C03649=1176.363,-28.044,-44.088,179.704,5.815,149.123
C03650=1176.358,-27.795,-44.101,179.705,5.815,149.122
C03651=1176.352,-27.545,-44.113,179.708,5.816,149.121
C03652=1176.347,-27.295,-44.125,179.711,5.816,149.121
C03653=1176.342,-27.046,-44.138,179.713,5.817,149.120
C03654=1176.337,-26.795,-44.150,179.715,5.817,149.120
C03655=1176.332,-26.546,-44.163,179.718,5.818,149.119
C03656=1176.327,-26.297,-44.175,179.720,5.819,149.118
C03657=1176.322,-26.047,-44.188,179.723,5.819,149.118
C03658=1176.316,-25.798,-44.200,179.725,5.819,149.117
C03659=1176.311,-25.548,-44.212,179.727,5.820,149.117
C03660=1176.307,-25.298,-44.225,179.730,5.820,149.116
C03661=1176.301,-25.048,-44.237,179.733,5.821,149.115
C03662=1176.296,-24.799,-44.250,179.735,5.821,149.115
C03663=1176.291,-24.550,-44.262,179.737,5.822,149.114
C03664=1176.286,-24.300,-44.275,179.740,5.822,149.113
C03665=1176.280,-24.030,-44.289,179.742,5.823,149.113
C03666=1176.275,-23.760,-44.302,179.745,5.824,149.112
C03667=1176.269,-23.491,-44.316,179.748,5.824,149.111
C03668=1176.264,-23.221,-44.330,179.750,5.824,149.111
C03669=1176.258,-22.971,-44.342,179.753,5.825,149.110
C03670=1176.253,-22.722,-44.354,179.755,5.826,149.110
C03671=1176.249,-22.472,-44.367,179.758,5.826,149.109
C03672=1176.243,-22.222,-44.380,179.760,5.826,149.108
C03673=1176.238,-21.973,-44.393,179.762,5.827,149.108
C03674=1176.232,-21.723,-44.405,179.765,5.827,149.107
C03675=1176.228,-21.473,-44.418,179.767,5.827,149.106
C03676=1176.223,-21.223,-44.431,179.769,5.828,149.106
C03677=1176.217,-20.974,-44.443,179.772,5.829,149.105
C03678=1176.212,-20.725,-44.456,179.775,5.829,149.104
C03679=1176.206,-20.475,-44.469,179.777,5.830,149.104
C03680=1176.202,-20.225,-44.482,179.780,5.830,149.103
C03681=1176.196,-19.975,-44.494,179.782,5.831,149.103
C03682=1176.191,-19.726,-44.506,179.784,5.831,149.102
C03683=1176.186,-19.477,-44.519,179.787,5.831,149.101
C03684=1176.181,-19.226,-44.533,179.789,5.832,149.101
C03685=1176.176,-18.977,-44.545,179.791,5.833,149.100
C03686=1176.171,-18.728,-44.558,179.794,5.833,149.100
C03687=1176.166,-18.478,-44.571,179.797,5.834,149.099
C03688=1176.161,-18.228,-44.583,179.799,5.834,149.098
C03689=1176.155,-17.979,-44.597,179.801,5.835,149.098
C03690=1176.150,-17.729,-44.609,179.804,5.835,149.097
C03691=1176.146,-17.479,-44.622,179.806,5.836,149.097
C03692=1176.140,-17.230,-44.635,179.809,5.837,149.096
C03693=1176.135,-16.980,-44.648,179.811,5.836,149.095
C03694=1176.130,-16.730,-44.661,179.813,5.837,149.095
C03695=1176.125,-16.481,-44.674,179.816,5.838,149.094
C03696=1176.119,-16.231,-44.687,179.819,5.838,149.093
C03697=1176.114,-15.982,-44.699,179.821,5.839,149.093
C03698=1176.109,-15.732,-44.712,179.823,5.839,149.092
C03699=1176.104,-15.483,-44.725,179.826,5.840,149.091
C03700=1176.098,-15.233,-44.738,179.828,5.841,149.091
C03701=1176.094,-14.983,-44.751,179.831,5.841,149.090
C03702=1176.089,-14.734,-44.764,179.834,5.841,149.090
C03703=1176.083,-14.484,-44.777,179.836,5.842,149.089
C03704=1176.078,-14.234,-44.790,179.838,5.843,149.088
C03705=1176.073,-13.985,-44.802,179.841,5.843,149.088
C03706=1176.067,-13.735,-44.816,179.843,5.844,149.087
C03707=1176.063,-13.485,-44.829,179.845,5.844,149.087
C03708=1176.058,-13.236,-44.841,179.848,5.844,149.086
C03709=1176.053,-12.986,-44.855,179.850,5.845,149.085
C03710=1176.048,-12.737,-44.868,179.853,5.845,149.085
C03711=1176.043,-12.487,-44.881,179.855,5.846,149.084
C03712=1176.037,-12.237,-44.894,179.858,5.847,149.084
C03713=1176.032,-11.988,-44.907,179.860,5.847,149.083
C03714=1176.027,-11.738,-44.919,179.863,5.848,149.082
C03715=1176.022,-11.488,-44.933,179.865,5.848,149.082
C03716=1176.017,-11.239,-44.946,179.868,5.849,149.081
C03717=1176.012,-10.989,-44.960,179.870,5.849,149.080
C03718=1176.007,-10.740,-44.972,179.873,5.850,149.080
C03719=1176.001,-10.490,-44.985,179.875,5.851,149.079
C03720=1175.996,-10.240,-44.999,179.878,5.851,149.078
C03721=1175.991,-9.991,-45.012,179.880,5.852,149.078
C03722=1175.986,-9.741,-45.025,179.883,5.852,149.077
C03723=1175.981,-9.492,-45.038,179.885,5.853,149.077
C03724=1175.976,-9.242,-45.051,179.888,5.854,149.076
C03725=1175.971,-8.992,-45.064,179.890,5.854,149.075
C03726=1175.966,-8.743,-45.078,179.893,5.855,149.075
C03727=1175.961,-8.493,-45.091,179.895,5.855,149.074
C03728=1175.955,-8.244,-45.104,179.897,5.855,149.074
C03729=1175.950,-7.994,-45.118,179.900,5.856,149.073
C03730=1175.945,-7.745,-45.131,179.902,5.856,149.072
C03731=1175.939,-7.495,-45.144,179.905,5.857,149.072
C03732=1175.935,-7.245,-45.157,179.907,5.857,149.071
C03733=1175.929,-6.996,-45.171,179.909,5.858,149.071
C03734=1175.925,-6.746,-45.184,179.912,5.859,149.070
C03735=1175.919,-6.496,-45.197,179.915,5.859,149.069
C03736=1175.915,-6.247,-45.211,179.917,5.860,149.069
C03737=1175.909,-5.997,-45.224,179.920,5.860,149.068
C03738=1175.904,-5.747,-45.237,179.922,5.861,149.067
C03739=1175.899,-5.498,-45.251,179.924,5.862,149.067
C03740=1175.894,-5.248,-45.264,179.927,5.862,149.066
C03741=1175.888,-4.999,-45.277,179.930,5.863,149.066
C03742=1175.884,-4.749,-45.290,179.932,5.863,149.065
C03743=1175.878,-4.500,-45.304,179.935,5.864,149.064
C03744=1175.874,-4.250,-45.317,179.937,5.864,149.064
C03745=1175.868,-4.001,-45.331,179.939,5.865,149.063
C03746=1175.864,-3.751,-45.343,179.942,5.866,149.063
C03747=1175.858,-3.502,-45.357,179.944,5.866,149.062
C03748=1175.853,-3.251,-45.371,179.947,5.867,149.061
C03749=1175.848,-3.003,-45.384,179.949,5.867,149.061
C03750=1175.843,-2.752,-45.398,179.952,5.868,149.060
C03751=1175.838,-2.504,-45.411,179.954,5.869,149.060
C03752=1175.833,-2.253,-45.425,179.957,5.869,149.059
C03753=1175.828,-2.005,-45.438,179.959,5.870,149.058
C03754=1175.823,-1.754,-45.452,179.962,5.870,149.058
C03755=1175.817,-1.505,-45.465,179.964,5.871,149.057
C03756=1175.813,-1.255,-45.478,179.967,5.872,149.057
C03757=1175.807,-1.006,-45.492,179.969,5.872,149.056
C03758=1175.802,-0.756,-45.506,179.972,5.873,149.055
C03759=1175.797,-0.507,-45.519,179.974,5.873,149.055
C03760=1175.792,-0.257,-45.533,179.977,5.874,149.054
C03761=1175.788,-0.007,-45.546,179.979,5.874,149.053
C03762=1175.782,0.242,-45.560,179.982,5.875,149.053
C03763=1175.777,0.492,-45.574,179.984,5.876,149.052
C03764=1175.772,0.741,-45.587,179.987,5.876,149.052
C03765=1175.767,0.991,-45.601,179.989,5.877,149.051
C03766=1175.761,1.241,-45.614,179.992,5.877,149.050
C03767=1175.756,1.490,-45.628,179.994,5.878,149.050
C03768=1175.752,1.740,-45.642,179.997,5.879,149.049
C03769=1175.745,2.009,-45.656,179.999,5.879,149.049
C03770=1175.740,2.278,-45.671,-179.998,5.880,149.048
C03771=1175.734,2.548,-45.686,-179.995,5.881,149.047
C03772=1175.729,2.817,-45.701,-179.992,5.881,149.046
C03773=1175.724,3.066,-45.714,-179.990,5.882,149.046
C03774=1175.719,3.316,-45.728,-179.987,5.883,149.045
C03775=1175.713,3.565,-45.742,-179.985,5.883,149.045
C03776=1175.708,3.815,-45.756,-179.983,5.884,149.044
C03777=1175.704,4.065,-45.769,-179.980,5.885,149.043
C03778=1175.698,4.314,-45.783,-179.977,5.885,149.043
C03779=1175.693,4.564,-45.797,-179.975,5.886,149.042
C03780=1175.688,4.813,-45.811,-179.972,5.886,149.042
C03781=1175.683,5.063,-45.824,-179.970,5.887,149.041
C03782=1175.678,5.312,-45.838,-179.968,5.888,149.040
C03783=1175.673,5.561,-45.852,-179.965,5.888,149.040
C03784=1175.668,5.812,-45.866,-179.962,5.889,149.039
C03785=1175.663,6.061,-45.879,-179.960,5.889,149.039
C03786=1175.658,6.310,-45.893,-179.958,5.890,149.038
C03787=1175.653,6.560,-45.908,-179.955,5.890,149.037
C03788=1175.648,6.810,-45.921,-179.953,5.891,149.037
C03789=1175.642,7.059,-45.935,-179.950,5.892,149.036
C03790=1175.638,7.309,-45.949,-179.948,5.893,149.036
C03791=1175.633,7.558,-45.963,-179.945,5.894,149.035
C03792=1175.627,7.807,-45.977,-179.942,5.894,149.034
C03793=1175.622,8.058,-45.991,-179.940,5.895,149.034
C03794=1175.617,8.307,-46.005,-179.937,5.896,149.033
C03795=1175.612,8.557,-46.019,-179.935,5.896,149.032
C03796=1175.607,8.806,-46.032,-179.932,5.897,149.032
C03797=1175.602,9.056,-46.047,-179.930,5.897,149.031
C03798=1175.597,9.306,-46.060,-179.927,5.898,149.031
C03799=1175.591,9.555,-46.074,-179.925,5.899,149.030
C03800=1175.587,9.805,-46.088,-179.922,5.899,149.030
C03801=1175.582,10.054,-46.103,-179.920,5.900,149.029
C03802=1175.576,10.303,-46.117,-179.917,5.900,149.028
C03803=1175.571,10.553,-46.131,-179.915,5.901,149.028
C03804=1175.566,10.803,-46.145,-179.912,5.901,149.027
C03805=1175.562,11.052,-46.159,-179.910,5.902,149.027
C03806=1175.556,11.301,-46.173,-179.907,5.903,149.026
C03807=1175.551,11.551,-46.186,-179.905,5.904,149.025
C03808=1175.546,11.801,-46.201,-179.902,5.905,149.025
C03809=1175.541,12.051,-46.215,-179.899,5.905,149.024
C03810=1175.536,12.300,-46.229,-179.897,5.906,149.024
C03811=1175.531,12.550,-46.243,-179.894,5.907,149.023
C03812=1175.526,12.799,-46.257,-179.892,5.907,149.022
C03813=1175.521,13.049,-46.272,-179.890,5.908,149.022
C03814=1175.515,13.298,-46.286,-179.887,5.908,149.021
C03815=1175.510,13.548,-46.300,-179.884,5.909,149.020
C03816=1175.505,13.797,-46.314,-179.882,5.910,149.020
C03817=1175.500,14.047,-46.328,-179.879,5.910,149.019
C03818=1175.495,14.297,-46.343,-179.877,5.911,149.019
C03819=1175.490,14.546,-46.357,-179.875,5.912,149.018
C03820=1175.485,14.796,-46.371,-179.871,5.913,149.017
C03821=1175.480,15.045,-46.385,-179.869,5.914,149.017
C03822=1175.475,15.295,-46.399,-179.867,5.914,149.016
C03823=1175.469,15.544,-46.413,-179.864,5.915,149.016
C03824=1175.464,15.794,-46.428,-179.862,5.916,149.015
C03825=1175.460,16.043,-46.443,-179.859,5.916,149.014
C03826=1175.455,16.293,-46.457,-179.857,5.916,149.014
C03827=1175.450,16.542,-46.471,-179.854,5.917,149.013
C03828=1175.445,16.792,-46.485,-179.852,5.918,149.013
C03829=1175.439,17.041,-46.499,-179.849,5.918,149.012
C03830=1175.434,17.291,-46.514,-179.847,5.919,149.011
C03831=1175.429,17.540,-46.528,-179.844,5.920,149.011
C03832=1175.424,17.790,-46.542,-179.841,5.921,149.010
C03833=1175.420,18.040,-46.556,-179.839,5.922,149.010
C03834=1175.415,18.289,-46.571,-179.836,5.922,149.009
C03835=1175.409,18.538,-46.585,-179.834,5.923,149.009
C03836=1175.404,18.788,-46.600,-179.831,5.924,149.008
C03837=1175.399,19.038,-46.614,-179.829,5.924,149.007
C03838=1175.394,19.287,-46.629,-179.827,5.925,149.007
C03839=1175.389,19.537,-46.643,-179.824,5.925,149.006
C03840=1175.384,19.786,-46.658,-179.821,5.927,149.005
C03841=1175.379,20.036,-46.672,-179.819,5.927,149.005
C03842=1175.374,20.286,-46.687,-179.816,5.928,149.004
C03843=1175.369,20.535,-46.700,-179.814,5.929,149.004
C03844=1175.363,20.784,-46.716,-179.811,5.929,149.003
C03845=1175.358,21.034,-46.730,-179.808,5.930,149.002
C03846=1175.353,21.283,-46.745,-179.806,5.931,149.002
C03847=1175.348,21.533,-46.759,-179.804,5.931,149.001
C03848=1175.344,21.782,-46.774,-179.800,5.932,149.001
C03849=1175.339,22.032,-46.788,-179.798,5.933,149.000
C03850=1175.333,22.282,-46.803,-179.796,5.934,148.999
C03851=1175.328,22.531,-46.818,-179.793,5.935,148.999
C03852=1175.324,22.781,-46.832,-179.791,5.935,148.998
C03853=1175.318,23.030,-46.846,-179.788,5.936,148.998
C03854=1175.313,23.279,-46.860,-179.786,5.936,148.997
C03855=1175.308,23.529,-46.876,-179.783,5.937,148.997
C03856=1175.303,23.779,-46.890,-179.780,5.938,148.996
C03857=1175.298,24.028,-46.905,-179.778,5.939,148.995
C03858=1175.293,24.277,-46.920,-179.775,5.940,148.995
C03859=1175.288,24.527,-46.934,-179.773,5.940,148.994
C03860=1175.283,24.776,-46.949,-179.770,5.941,148.994
C03861=1175.278,25.026,-46.964,-179.768,5.941,148.993
C03862=1175.273,25.276,-46.978,-179.766,5.942,148.992
C03863=1175.268,25.525,-46.993,-179.762,5.944,148.992
C03864=1175.262,25.775,-47.008,-179.760,5.944,148.991
C03865=1175.258,26.024,-47.023,-179.758,5.945,148.991
C03866=1175.253,26.274,-47.037,-179.755,5.945,148.990
C03867=1175.247,26.524,-47.052,-179.753,5.946,148.989
C03868=1175.243,26.773,-47.067,-179.750,5.947,148.989
C03869=1175.238,27.023,-47.081,-179.747,5.948,148.988
C03870=1175.233,27.272,-47.096,-179.745,5.949,148.988
C03871=1175.227,27.522,-47.111,-179.742,5.949,148.987
C03872=1175.223,27.771,-47.126,-179.740,5.950,148.987
C03873=1175.217,28.040,-47.142,-179.737,5.951,148.986
C03874=1175.212,28.309,-47.158,-179.734,5.952,148.985
C03875=1175.206,28.578,-47.174,-179.731,5.952,148.985
C03876=1175.201,28.847,-47.190,-179.729,5.953,148.984
C03877=1175.196,29.096,-47.205,-179.726,5.955,148.983
C03878=1175.191,29.345,-47.219,-179.723,5.955,148.983
C03879=1175.186,29.595,-47.235,-179.721,5.956,148.982
C03880=1175.181,29.845,-47.249,-179.719,5.956,148.982
C03881=1175.176,30.094,-47.264,-179.716,5.957,148.981
C03882=1175.170,30.344,-47.279,-179.714,5.958,148.980
C03883=1175.166,30.593,-47.294,-179.710,5.959,148.980
C03884=1175.160,30.842,-47.310,-179.708,5.960,148.979
C03885=1175.155,31.092,-47.324,-179.706,5.960,148.979
C03886=1175.151,31.341,-47.339,-179.703,5.961,148.978
C03887=1175.145,31.591,-47.354,-179.701,5.962,148.978
C03888=1175.140,31.840,-47.369,-179.698,5.963,148.977
C03889=1175.135,32.089,-47.384,-179.695,5.964,148.976
C03890=1175.130,32.339,-47.399,-179.693,5.964,148.976
C03891=1175.125,32.588,-47.414,-179.690,5.965,148.975
C03892=1175.120,32.838,-47.429,-179.688,5.966,148.975
C03893=1175.116,33.088,-47.444,-179.685,5.966,148.974
C03894=1175.110,33.337,-47.460,-179.682,5.968,148.973
C03895=1175.106,33.587,-47.475,-179.680,5.968,148.973
C03896=1175.100,33.837,-47.489,-179.677,5.969,148.972
C03897=1175.095,34.086,-47.504,-179.675,5.969,148.971
C03898=1175.090,34.335,-47.520,-179.673,5.970,148.971
C03899=1175.085,34.585,-47.534,-179.669,5.972,148.970
C03900=1175.079,34.834,-47.550,-179.667,5.972,148.970
C03901=1175.075,35.083,-47.565,-179.665,5.973,148.969
C03902=1175.069,35.333,-47.580,-179.662,5.973,148.969
C03903=1175.065,35.583,-47.595,-179.660,5.974,148.968
C03904=1175.060,35.833,-47.611,-179.656,5.976,148.967
C03905=1175.055,36.082,-47.626,-179.654,5.976,148.967
C03906=1175.050,36.331,-47.641,-179.652,5.977,148.966
C03907=1175.045,36.580,-47.656,-179.650,5.978,148.966
C03908=1175.039,36.830,-47.671,-179.646,5.979,148.965
C03909=1175.035,37.079,-47.686,-179.644,5.980,148.964
C03910=1175.030,37.329,-47.702,-179.642,5.980,148.964
C03911=1175.025,37.578,-47.717,-179.639,5.981,148.963
C03912=1175.020,37.828,-47.733,-179.637,5.982,148.963
C03913=1175.014,38.078,-47.748,-179.633,5.983,148.962
C03914=1175.010,38.327,-47.763,-179.631,5.984,148.962
C03915=1175.004,38.576,-47.778,-179.629,5.984,148.961
C03916=1175.000,38.826,-47.793,-179.626,5.985,148.960
C03917=1174.995,39.076,-47.809,-179.623,5.987,148.960
C03918=1174.989,39.325,-47.825,-179.621,5.987,148.959
C03919=1174.985,39.574,-47.840,-179.618,5.988,148.959
C03920=1174.979,39.823,-47.855,-179.616,5.989,148.958
C03921=1174.975,40.073,-47.871,-179.613,5.989,148.958
C03922=1174.970,40.323,-47.885,-179.610,5.991,148.957
C03923=1174.964,40.573,-47.901,-179.608,5.991,148.956
C03924=1174.960,40.822,-47.916,-179.605,5.992,148.956
C03925=1174.954,41.071,-47.932,-179.603,5.993,148.955
C03926=1174.949,41.321,-47.948,-179.600,5.994,148.955
C03927=1174.945,41.570,-47.963,-179.598,5.995,148.954
C03928=1174.939,41.820,-47.978,-179.595,5.995,148.954
C03929=1174.934,42.069,-47.994,-179.593,5.996,148.953
C03930=1174.930,42.319,-48.009,-179.590,5.997,148.952
C03931=1174.924,42.568,-48.025,-179.587,5.998,148.952
C03932=1174.919,42.818,-48.040,-179.585,5.999,148.951
C03933=1174.914,43.067,-48.055,-179.582,5.999,148.951
C03934=1174.910,43.317,-48.071,-179.579,6.001,148.950
C03935=1174.904,43.566,-48.087,-179.577,6.001,148.949
C03936=1174.899,43.816,-48.102,-179.575,6.002,148.949
C03937=1174.894,44.065,-48.117,-179.572,6.003,148.948
C03938=1174.890,44.314,-48.134,-179.569,6.004,148.948
C03939=1174.884,44.564,-48.150,-179.567,6.005,148.947
C03940=1174.880,44.813,-48.165,-179.564,6.005,148.947
C03941=1174.874,45.062,-48.180,-179.562,6.006,148.946
C03942=1174.870,45.312,-48.196,-179.559,6.008,148.945
C03943=1174.864,45.562,-48.212,-179.556,6.009,148.945
C03944=1174.860,45.811,-48.227,-179.554,6.009,148.944
C03945=1174.855,46.061,-48.243,-179.551,6.010,148.944
C03946=1174.849,46.310,-48.258,-179.548,6.011,148.943
C03947=1174.844,46.559,-48.275,-179.546,6.012,148.943
C03948=1174.839,46.809,-48.291,-179.544,6.013,148.942
C03949=1174.835,47.058,-48.306,-179.540,6.014,148.941
C03950=1174.829,47.308,-48.321,-179.538,6.015,148.941
C03951=1174.825,47.558,-48.337,-179.536,6.015,148.940
C03952=1174.819,47.807,-48.353,-179.533,6.016,148.940
C03953=1174.814,48.056,-48.369,-179.530,6.017,148.939
C03954=1174.810,48.306,-48.384,-179.528,6.018,148.939
C03955=1174.805,48.555,-48.400,-179.525,6.019,148.938
C03956=1174.799,48.805,-48.416,-179.522,6.020,148.937
C03957=1174.795,49.054,-48.432,-179.520,6.021,148.937
C03958=1174.789,49.303,-48.448,-179.517,6.021,148.936
C03959=1174.784,49.553,-48.463,-179.515,6.022,148.936
C03960=1174.780,49.803,-48.479,-179.512,6.024,148.935
C03961=1174.775,50.051,-48.495,-179.509,6.024,148.935
C03962=1174.770,50.301,-48.511,-179.507,6.025,148.934
C03963=1174.765,50.551,-48.527,-179.504,6.026,148.933
C03964=1174.760,50.800,-48.543,-179.502,6.027,148.933
C03965=1174.755,51.050,-48.559,-179.499,6.028,148.932
C03966=1174.750,51.299,-48.574,-179.496,6.029,148.932
C03967=1174.744,51.548,-48.591,-179.494,6.030,148.931
C03968=1174.740,51.798,-48.607,-179.491,6.030,148.931
C03969=1174.735,52.047,-48.622,-179.489,6.031,148.930
C03970=1174.731,52.297,-48.638,-179.486,6.033,148.929
C03971=1174.725,52.546,-48.654,-179.484,6.033,148.929
C03972=1174.720,52.795,-48.670,-179.481,6.034,148.928
C03973=1174.715,53.045,-48.686,-179.478,6.036,148.928
C03974=1174.710,53.294,-48.702,-179.476,6.036,148.927
C03975=1174.705,53.544,-48.718,-179.474,6.037,148.927
C03976=1174.700,53.793,-48.734,-179.470,6.038,148.926
C03977=1174.694,54.062,-48.751,-179.468,6.039,148.925
C03978=1174.690,54.331,-48.768,-179.465,6.041,148.925
C03979=1174.684,54.599,-48.786,-179.462,6.041,148.924
C03980=1174.679,54.867,-48.803,-179.459,6.042,148.924
C03981=1174.674,55.117,-48.819,-179.457,6.043,148.923
C03982=1174.669,55.366,-48.835,-179.454,6.044,148.923
C03983=1174.664,55.616,-48.851,-179.452,6.045,148.922
C03984=1174.659,55.865,-48.868,-179.449,6.046,148.922
C03985=1174.654,56.114,-48.883,-179.446,6.046,148.921
C03986=1174.649,56.364,-48.900,-179.444,6.048,148.920
C03987=1174.643,56.614,-48.916,-179.441,6.049,148.920
C03988=1174.639,56.863,-48.933,-179.439,6.050,148.919
C03989=1174.633,57.113,-48.948,-179.436,6.051,148.919
C03990=1174.629,57.362,-48.965,-179.433,6.052,148.918
C03991=1174.623,57.611,-48.981,-179.431,6.052,148.918
C03992=1174.619,57.861,-48.997,-179.428,6.054,148.917
C03993=1174.614,58.110,-49.014,-179.425,6.054,148.916
C03994=1174.609,58.360,-49.030,-179.423,6.055,148.916
C03995=1174.604,58.609,-49.046,-179.420,6.057,148.915
C03996=1174.599,58.859,-49.062,-179.418,6.058,148.915
C03997=1174.594,59.107,-49.078,-179.415,6.058,148.914
C03998=1174.589,59.357,-49.095,-179.412,6.060,148.914
C03999=1174.583,59.607,-49.111,-179.410,6.060,148.913
C04000=1174.579,59.856,-49.128,-179.407,6.061,148.912
C04001=1174.574,60.106,-49.144,-179.404,6.062,148.912
C04002=1174.569,60.355,-49.160,-179.402,6.063,148.911
C04003=1174.565,60.604,-49.177,-179.399,6.065,148.911
C04004=1174.559,60.854,-49.192,-179.396,6.065,148.910
C04005=1174.555,61.103,-49.209,-179.394,6.066,148.910
C04006=1174.549,61.352,-49.226,-179.391,6.067,148.909
C04007=1174.544,61.602,-49.242,-179.389,6.068,148.909
C04008=1174.539,61.851,-49.258,-179.386,6.069,148.908
C04009=1174.534,62.101,-49.275,-179.384,6.070,148.908
C04010=1174.530,62.350,-49.291,-179.381,6.071,148.907
C04011=1174.525,62.599,-49.308,-179.379,6.072,148.907
C04012=1174.519,62.850,-49.324,-179.376,6.073,148.906
C04013=1174.514,63.098,-49.341,-179.373,6.074,148.905
C04014=1174.510,63.348,-49.357,-179.370,6.075,148.905
C04015=1174.505,63.597,-49.373,-179.368,6.076,148.904
C04016=1174.499,63.847,-49.390,-179.365,6.077,148.904
C04017=1174.495,64.096,-49.407,-179.363,6.078,148.903
C04018=1174.490,64.345,-49.423,-179.360,6.079,148.903
C04019=1174.485,64.595,-49.440,-179.357,6.081,148.902
C04020=1174.481,64.844,-49.456,-179.355,6.081,148.902
C04021=1174.475,65.094,-49.473,-179.353,6.082,148.901
C04022=1174.470,65.343,-49.489,-179.349,6.083,148.900
C04023=1174.465,65.592,-49.505,-179.347,6.084,148.900
C04024=1174.460,65.842,-49.523,-179.345,6.085,148.899
C04025=1174.455,66.091,-49.539,-179.342,6.086,148.899
C04026=1174.450,66.340,-49.556,-179.339,6.087,148.898
C04027=1174.446,66.590,-49.572,-179.336,6.089,148.898
C04028=1174.441,66.840,-49.590,-179.334,6.089,148.897
C04029=1174.435,67.088,-49.606,-179.332,6.090,148.897
C04030=1174.431,67.338,-49.622,-179.328,6.091,148.896
C04031=1174.425,67.588,-49.639,-179.326,6.092,148.896
C04032=1174.420,67.837,-49.655,-179.323,6.094,148.895
C04033=1174.416,68.086,-49.672,-179.321,6.095,148.895
C04034=1174.411,68.336,-49.689,-179.318,6.095,148.894
C04035=1174.406,68.585,-49.706,-179.316,6.097,148.893
C04036=1174.401,68.835,-49.722,-179.313,6.097,148.893
C04037=1174.396,69.084,-49.740,-179.310,6.099,148.892
C04038=1174.391,69.334,-49.756,-179.308,6.099,148.892
C04039=1174.386,69.583,-49.773,-179.305,6.101,148.891
C04040=1174.381,69.832,-49.790,-179.302,6.102,148.891
C04041=1174.377,70.082,-49.807,-179.300,6.103,148.890
C04042=1174.371,70.331,-49.823,-179.297,6.104,148.889
C04043=1174.366,70.580,-49.840,-179.295,6.105,148.889
C04044=1174.362,70.830,-49.857,-179.292,6.106,148.888
C04045=1174.356,71.079,-49.874,-179.289,6.107,148.888
C04046=1174.352,71.328,-49.891,-179.286,6.108,148.887
C04047=1174.347,71.578,-49.908,-179.284,6.109,148.887
C04048=1174.342,71.827,-49.925,-179.281,6.110,148.886
C04049=1174.336,72.076,-49.942,-179.279,6.111,148.886
C04050=1174.332,72.326,-49.959,-179.276,6.112,148.885
C04051=1174.327,72.576,-49.976,-179.273,6.114,148.885
C04052=1174.322,72.825,-49.993,-179.271,6.114,148.884
C04053=1174.317,73.074,-50.009,-179.268,6.116,148.884
C04054=1174.312,73.324,-50.026,-179.266,6.117,148.883
C04055=1174.308,73.572,-50.043,-179.263,6.117,148.883
C04056=1174.303,73.822,-50.061,-179.260,6.119,148.882
C04057=1174.298,74.072,-50.077,-179.258,6.120,148.881
C04058=1174.292,74.321,-50.094,-179.255,6.121,148.881
C04059=1174.288,74.570,-50.111,-179.252,6.122,148.880
C04060=1174.283,74.820,-50.129,-179.250,6.123,148.880
C04061=1174.278,75.069,-50.146,-179.247,6.124,148.879
C04062=1174.273,75.319,-50.163,-179.244,6.126,148.879
C04063=1174.267,75.568,-50.180,-179.242,6.126,148.878
C04064=1174.263,75.817,-50.197,-179.240,6.127,148.878
C04065=1174.258,76.067,-50.214,-179.236,6.128,148.877
C04066=1174.253,76.316,-50.231,-179.234,6.129,148.877
C04067=1174.248,76.566,-50.248,-179.231,6.131,148.876
C04068=1174.243,76.814,-50.265,-179.229,6.132,148.876
C04069=1174.238,77.064,-50.283,-179.226,6.133,148.875
C04070=1174.234,77.313,-50.299,-179.224,6.134,148.875
C04071=1174.229,77.562,-50.317,-179.221,6.135,148.874
C04072=1174.224,77.812,-50.335,-179.218,6.136,148.873
C04073=1174.219,78.062,-50.351,-179.215,6.138,148.873
C04074=1174.214,78.310,-50.369,-179.213,6.138,148.872
C04075=1174.209,78.560,-50.386,-179.210,6.140,148.872
C04076=1174.204,78.809,-50.403,-179.207,6.140,148.871
C04077=1174.199,79.059,-50.421,-179.205,6.142,148.871
C04078=1174.195,79.308,-50.437,-179.202,6.143,148.870
C04079=1174.189,79.558,-50.455,-179.199,6.144,148.870
C04080=1174.184,79.807,-50.473,-179.197,6.145,148.869
C04081=1174.179,80.075,-50.490,-179.194,6.147,148.869
C04082=1174.174,80.344,-50.509,-179.191,6.147,148.868
C04083=1174.169,80.612,-50.529,-179.189,6.149,148.868
C04084=1174.163,80.880,-50.547,-179.185,6.150,148.867
C04085=1174.158,81.130,-50.564,-179.183,6.151,148.867
C04086=1174.153,81.379,-50.581,-179.180,6.152,148.866
C04087=1174.148,81.629,-50.599,-179.178,6.153,148.865
C04088=1174.144,81.878,-50.616,-179.175,6.155,148.865
C04089=1174.139,82.127,-50.633,-179.173,6.156,148.864
C04090=1174.134,82.377,-50.651,-179.169,6.157,148.864
C04091=1174.129,82.626,-50.669,-179.167,6.158,148.863
C04092=1174.124,82.875,-50.686,-179.165,6.159,148.863
C04093=1174.119,83.125,-50.703,-179.162,6.160,148.862
C04094=1174.114,83.374,-50.721,-179.159,6.162,148.862
C04095=1174.109,83.623,-50.739,-179.157,6.162,148.861
C04096=1174.105,83.873,-50.756,-179.154,6.164,148.861
C04097=1174.099,84.121,-50.774,-179.151,6.164,148.860
C04098=1174.094,84.371,-50.791,-179.148,6.166,148.860
C04099=1174.089,84.620,-50.809,-179.146,6.167,148.859
C04100=1174.085,84.870,-50.825,-179.143,6.168,148.859
C04101=1174.080,85.119,-50.843,-179.141,6.169,148.858
C04102=1174.075,85.368,-50.861,-179.138,6.171,148.858
C04103=1174.070,85.618,-50.879,-179.136,6.172,148.857
C04104=1174.065,85.867,-50.897,-179.132,6.173,148.856
C04105=1174.061,86.116,-50.914,-179.130,6.174,148.856
C04106=1174.055,86.366,-50.931,-179.128,6.176,148.856
C04107=1174.050,86.615,-50.949,-179.125,6.176,148.855
C04108=1174.046,86.864,-50.967,-179.122,6.178,148.855
C04109=1174.040,87.114,-50.985,-179.120,6.178,148.854
C04110=1174.035,87.363,-51.003,-179.117,6.180,148.853
C04111=1174.031,87.612,-51.020,-179.115,6.181,148.853
C04112=1174.026,87.862,-51.037,-179.112,6.182,148.852
C04113=1174.021,88.111,-51.055,-179.109,6.184,148.852
C04114=1174.016,88.360,-51.073,-179.106,6.184,148.851
C04115=1174.011,88.609,-51.091,-179.103,6.186,148.851
C04116=1174.006,88.859,-51.108,-179.101,6.187,148.850
C04117=1174.001,89.108,-51.126,-179.098,6.188,148.850
C04118=1173.997,89.358,-51.145,-179.096,6.189,148.849
C04119=1173.992,89.607,-51.163,-179.093,6.191,148.849
C04120=1173.987,89.857,-51.180,-179.091,6.192,148.848
C04121=1173.982,90.106,-51.198,-179.087,6.193,148.848
C04122=1173.978,90.355,-51.215,-179.085,6.194,148.847
C04123=1173.973,90.604,-51.233,-179.083,6.196,148.847
C04124=1173.968,90.853,-51.251,-179.079,6.197,148.846
C04125=1173.963,91.103,-51.269,-179.077,6.198,148.846
C04126=1173.958,91.352,-51.287,-179.074,6.199,148.845
C04127=1173.953,91.602,-51.304,-179.072,6.200,148.845
C04128=1173.948,91.851,-51.322,-179.069,6.202,148.844
C04129=1173.943,92.100,-51.340,-179.067,6.202,148.844
C04130=1173.938,92.349,-51.358,-179.064,6.204,148.843
C04131=1173.934,92.599,-51.377,-179.062,6.205,148.843
C04132=1173.929,92.848,-51.395,-179.058,6.206,148.842
C04133=1173.924,93.097,-51.413,-179.056,6.208,148.842
C04134=1173.919,93.347,-51.431,-179.053,6.208,148.841
C04135=1173.914,93.596,-51.449,-179.050,6.210,148.841
C04136=1173.909,93.846,-51.466,-179.048,6.211,148.840
C04137=1173.904,94.095,-51.484,-179.045,6.212,148.840
C04138=1173.899,94.344,-51.502,-179.043,6.213,148.839
C04139=1173.895,94.594,-51.520,-179.040,6.215,148.839
C04140=1173.889,94.843,-51.539,-179.037,6.216,148.838
C04141=1173.884,95.092,-51.557,-179.035,6.217,148.838
C04142=1173.879,95.342,-51.575,-179.032,6.219,148.837
C04143=1173.874,95.591,-51.593,-179.030,6.220,148.837
C04144=1173.869,95.840,-51.611,-179.027,6.221,148.836
C04145=1173.865,96.089,-51.629,-179.024,6.223,148.836
C04146=1173.861,96.338,-51.648,-179.021,6.224,148.835
C04147=1173.856,96.588,-51.666,-179.018,6.225,148.835
C04148=1173.851,96.837,-51.684,-179.016,6.226,148.834
C04149=1173.846,97.086,-51.702,-179.013,6.228,148.834
C04150=1173.841,97.335,-51.720,-179.010,6.229,148.833
C04151=1173.836,97.585,-51.739,-179.008,6.230,148.833
C04152=1173.831,97.834,-51.757,-179.005,6.231,148.832
C04153=1173.826,98.084,-51.775,-179.003,6.232,148.832
C04154=1173.821,98.333,-51.793,-179.000,6.234,148.831
C04155=1173.816,98.582,-51.811,-178.997,6.235,148.831
C04156=1173.812,98.831,-51.830,-178.995,6.236,148.830
C04157=1173.807,99.081,-51.848,-178.992,6.238,148.830
C04158=1173.802,99.330,-51.866,-178.989,6.238,148.829
C04159=1173.797,99.579,-51.884,-178.987,6.240,148.829
C04160=1173.792,99.828,-51.902,-178.984,6.242,148.828
C04161=1173.788,100.078,-51.921,-178.981,6.242,148.828
C04162=1173.782,100.327,-51.940,-178.979,6.244,148.827
C04163=1173.777,100.576,-51.958,-178.976,6.245,148.827
C04164=1173.772,100.825,-51.976,-178.973,6.246,148.826
C04165=1173.768,101.075,-51.994,-178.971,6.248,148.826
C04166=1173.763,101.324,-52.013,-178.968,6.249,148.825
C04167=1173.758,101.573,-52.031,-178.965,6.250,148.825
C04168=1173.753,101.823,-52.050,-178.962,6.252,148.824
C04169=1173.749,102.072,-52.068,-178.960,6.253,148.824
C04170=1173.744,102.321,-52.086,-178.957,6.254,148.823
C04171=1173.738,102.570,-52.105,-178.955,6.255,148.823
C04172=1173.734,102.820,-52.123,-178.952,6.257,148.822
C04173=1173.729,103.069,-52.142,-178.949,6.258,148.822
C04174=1173.724,103.318,-52.161,-178.947,6.259,148.821
C04175=1173.719,103.567,-52.179,-178.944,6.261,148.821
C04176=1173.715,103.817,-52.198,-178.941,6.262,148.820
C04177=1173.709,104.066,-52.216,-178.939,6.263,148.820
C04178=1173.705,104.315,-52.235,-178.936,6.265,148.819
C04179=1173.700,104.565,-52.253,-178.933,6.266,148.819
C04180=1173.695,104.814,-52.272,-178.931,6.267,148.818
C04181=1173.690,105.063,-52.290,-178.928,6.269,148.818
C04182=1173.686,105.313,-52.309,-178.925,6.270,148.817
C04183=1173.680,105.561,-52.328,-178.923,6.271,148.817
C04184=1173.675,105.811,-52.346,-178.920,6.273,148.817
C04185=1173.671,106.080,-52.366,-178.917,6.274,148.816
C04186=1173.665,106.347,-52.387,-178.914,6.276,148.816
C04187=1173.660,106.616,-52.407,-178.912,6.276,148.815
C04188=1173.655,106.885,-52.426,-178.909,6.278,148.814
C04189=1173.650,107.134,-52.446,-178.906,6.279,148.814
C04190=1173.645,107.383,-52.464,-178.903,6.281,148.813
C04191=1173.641,107.632,-52.483,-178.901,6.282,148.813
C04192=1173.635,107.882,-52.501,-178.898,6.283,148.812
C04193=1173.631,108.130,-52.520,-178.895,6.285,148.812
C04194=1173.626,108.380,-52.540,-178.893,6.286,148.812
C04195=1173.621,108.629,-52.558,-178.890,6.288,148.811
C04196=1173.616,108.879,-52.577,-178.887,6.289,148.811
C04197=1173.611,109.128,-52.595,-178.885,6.290,148.810
C04198=1173.607,109.376,-52.614,-178.882,6.292,148.810
C04199=1173.602,109.627,-52.633,-178.879,6.293,148.809
C04200=1173.597,109.875,-52.652,-178.877,6.294,148.809
C04201=1173.592,110.125,-52.671,-178.874,6.296,148.808
C04202=1173.587,110.374,-52.689,-178.871,6.297,148.808
C04203=1173.582,110.623,-52.709,-178.869,6.298,148.807
C04204=1173.578,110.873,-52.727,-178.866,6.300,148.807
C04205=1173.572,111.122,-52.746,-178.863,6.302,148.806
C04206=1173.568,111.371,-52.765,-178.861,6.302,148.806
C04207=1173.563,111.620,-52.784,-178.858,6.304,148.805
C04208=1173.559,111.870,-52.803,-178.855,6.306,148.805
C04209=1173.553,112.118,-52.822,-178.852,6.307,148.804
C04210=1173.549,112.368,-52.842,-178.850,6.308,148.804
C04211=1173.544,112.617,-52.860,-178.847,6.310,148.803
C04212=1173.538,112.866,-52.879,-178.844,6.311,148.803
C04213=1173.534,113.115,-52.898,-178.842,6.312,148.802
C04214=1173.529,113.365,-52.917,-178.839,6.314,148.802
C04215=1173.525,113.614,-52.936,-178.836,6.315,148.802
C04216=1173.519,113.863,-52.955,-178.834,6.316,148.801
C04217=1173.515,114.112,-52.975,-178.831,6.318,148.801
C04218=1173.510,114.362,-52.993,-178.828,6.319,148.800
C04219=1173.505,114.611,-53.012,-178.826,6.321,148.800
C04220=1173.500,114.860,-53.032,-178.823,6.322,148.799
C04221=1173.496,115.109,-53.051,-178.820,6.323,148.799
C04222=1173.490,115.358,-53.070,-178.818,6.325,148.798
C04223=1173.486,115.607,-53.089,-178.815,6.326,148.798
C04224=1173.481,115.857,-53.108,-178.812,6.327,148.797
C04225=1173.476,116.106,-53.127,-178.810,6.329,148.797
C04226=1173.471,116.355,-53.146,-178.807,6.331,148.797
C04227=1173.466,116.605,-53.166,-178.804,6.331,148.796
C04228=1173.462,116.854,-53.185,-178.802,6.333,148.795
C04229=1173.457,117.103,-53.204,-178.799,6.335,148.795
C04230=1173.452,117.352,-53.224,-178.796,6.337,148.795
C04231=1173.447,117.601,-53.243,-178.794,6.337,148.794
C04232=1173.442,117.851,-53.263,-178.791,6.339,148.794
C04233=1173.437,118.100,-53.281,-178.788,6.341,148.793
C04234=1173.433,118.349,-53.300,-178.785,6.342,148.793
C04235=1173.427,118.598,-53.320,-178.783,6.343,148.792
C04236=1173.423,118.848,-53.339,-178.780,6.345,148.792
C04237=1173.419,119.097,-53.358,-178.777,6.346,148.791
C04238=1173.413,119.346,-53.378,-178.775,6.347,148.791
C04239=1173.408,119.596,-53.397,-178.772,6.349,148.790
C04240=1173.404,119.844,-53.416,-178.769,6.350,148.790
C04241=1173.399,120.094,-53.436,-178.767,6.352,148.790
C04242=1173.394,120.343,-53.455,-178.765,6.353,148.789
C04243=1173.389,120.592,-53.474,-178.761,6.354,148.789
C04244=1173.385,120.841,-53.495,-178.759,6.356,148.788
C04245=1173.380,121.090,-53.514,-178.756,6.358,148.788
C04246=1173.375,121.339,-53.533,-178.753,6.360,148.787
C04247=1173.371,121.589,-53.553,-178.751,6.360,148.787
C04248=1173.365,121.838,-53.572,-178.748,6.362,148.786
C04249=1173.360,122.087,-53.592,-178.745,6.364,148.786
C04250=1173.356,122.336,-53.611,-178.742,6.365,148.785
C04251=1173.351,122.585,-53.630,-178.740,6.366,148.785
C04252=1173.346,122.835,-53.650,-178.737,6.368,148.784
C04253=1173.342,123.085,-53.669,-178.734,6.369,148.784
C04254=1173.337,123.333,-53.689,-178.732,6.371,148.784
C04255=1173.332,123.582,-53.709,-178.730,6.372,148.783
C04256=1173.327,123.832,-53.729,-178.727,6.374,148.783
C04257=1173.322,124.080,-53.747,-178.724,6.375,148.782
C04258=1173.318,124.330,-53.767,-178.721,6.377,148.782
C04259=1173.313,124.579,-53.788,-178.718,6.379,148.781
C04260=1173.308,124.828,-53.807,-178.716,6.379,148.781
C04261=1173.303,125.077,-53.826,-178.713,6.381,148.780
C04262=1173.298,125.327,-53.846,-178.710,6.383,148.780
C04263=1173.293,125.575,-53.866,-178.708,6.384,148.780
C04264=1173.289,125.825,-53.886,-178.705,6.385,148.779
C04265=1173.284,126.074,-53.905,-178.703,6.387,148.779
C04266=1173.279,126.324,-53.925,-178.700,6.388,148.778
C04267=1173.274,126.572,-53.945,-178.697,6.390,148.778
C04268=1173.270,126.821,-53.964,-178.694,6.392,148.777
C04269=1173.265,127.071,-53.984,-178.692,6.393,148.777
C04270=1173.260,127.319,-54.004,-178.689,6.394,148.777
C04271=1173.256,127.569,-54.023,-178.686,6.396,148.776
C04272=1173.251,127.818,-54.043,-178.683,6.398,148.776
C04273=1173.246,128.067,-54.064,-178.681,6.399,148.775
C04274=1173.241,128.316,-54.083,-178.679,6.400,148.775
C04275=1173.236,128.566,-54.102,-178.676,6.402,148.774
C04276=1173.232,128.815,-54.123,-178.673,6.403,148.774
C04277=1173.227,129.064,-54.142,-178.670,6.405,148.773
C04278=1173.222,129.313,-54.162,-178.667,6.407,148.773
C04279=1173.217,129.562,-54.182,-178.665,6.409,148.773
C04280=1173.212,129.812,-54.202,-178.662,6.410,148.772
C04281=1173.207,130.061,-54.223,-178.659,6.411,148.772
C04282=1173.203,130.310,-54.242,-178.657,6.413,148.771
C04283=1173.198,130.559,-54.262,-178.654,6.414,148.771
C04284=1173.193,130.808,-54.282,-178.651,6.416,148.770
C04285=1173.189,131.057,-54.302,-178.649,6.417,148.770
C04286=1173.184,131.307,-54.322,-178.646,6.419,148.770
C04287=1173.179,131.556,-54.342,-178.643,6.420,148.769
C04288=1173.174,131.805,-54.362,-178.640,6.422,148.769
C04289=1173.169,132.073,-54.384,-178.638,6.424,148.768
C04290=1173.164,132.342,-54.405,-178.635,6.425,148.768
C04291=1173.158,132.611,-54.427,-178.632,6.427,148.767
C04292=1173.153,132.879,-54.449,-178.629,6.428,148.767
C04293=1173.149,133.128,-54.468,-178.626,6.430,148.766
C04294=1173.144,133.377,-54.489,-178.624,6.432,148.766
C04295=1173.139,133.627,-54.509,-178.621,6.433,148.765
C04296=1173.134,133.876,-54.529,-178.618,6.435,148.765
C04297=1173.130,134.125,-54.550,-178.616,6.436,148.765
C04298=1173.125,134.374,-54.569,-178.613,6.438,148.764
C04299=1173.120,134.623,-54.589,-178.610,6.440,148.764
C04300=1173.116,134.872,-54.610,-178.608,6.441,148.763
C04301=1173.110,135.122,-54.630,-178.605,6.443,148.763
C04302=1173.106,135.370,-54.650,-178.602,6.444,148.762
C04303=1173.101,135.619,-54.671,-178.599,6.446,148.762
C04304=1173.097,135.869,-54.690,-178.597,6.447,148.762
C04305=1173.091,136.118,-54.711,-178.594,6.449,148.761
C04306=1173.087,136.367,-54.732,-178.592,6.451,148.761
C04307=1173.082,136.617,-54.751,-178.589,6.452,148.760
C04308=1173.077,136.865,-54.771,-178.586,6.454,148.760
C04309=1173.072,137.114,-54.792,-178.583,6.455,148.759
C04310=1173.068,137.363,-54.813,-178.580,6.457,148.759
C04311=1173.063,137.613,-54.832,-178.578,6.458,148.759
C04312=1173.058,137.862,-54.853,-178.575,6.460,148.758
C04313=1173.053,138.111,-54.874,-178.573,6.462,148.758
C04314=1173.049,138.360,-54.894,-178.570,6.463,148.758
C04315=1173.044,138.609,-54.915,-178.567,6.465,148.757
C04316=1173.039,138.859,-54.935,-178.564,6.466,148.757
C04317=1173.034,139.108,-54.955,-178.562,6.468,148.756
C04318=1173.030,139.357,-54.976,-178.559,6.470,148.756
C04319=1173.025,139.606,-54.996,-178.557,6.471,148.755
C04320=1173.020,139.855,-55.017,-178.554,6.473,148.755
C04321=1173.016,140.104,-55.037,-178.551,6.474,148.755
C04322=1173.011,140.353,-55.058,-178.549,6.476,148.754
C04323=1173.006,140.603,-55.078,-178.546,6.478,148.754
C04324=1173.002,140.852,-55.098,-178.543,6.479,148.753
C04325=1172.996,141.101,-55.119,-178.540,6.481,148.753
C04326=1172.992,141.350,-55.140,-178.537,6.483,148.752
C04327=1172.988,141.599,-55.160,-178.535,6.484,148.752
C04328=1172.982,141.848,-55.181,-178.532,6.486,148.752
C04329=1172.978,142.097,-55.201,-178.530,6.487,148.751
C04330=1172.973,142.346,-55.222,-178.527,6.489,148.751
C04331=1172.968,142.595,-55.243,-178.524,6.491,148.750
C04332=1172.964,142.844,-55.263,-178.522,6.492,148.750
C04333=1172.959,143.093,-55.284,-178.519,6.494,148.750
C04334=1172.954,143.342,-55.304,-178.516,6.495,148.749
C04335=1172.949,143.592,-55.325,-178.513,6.497,148.749
C04336=1172.945,143.841,-55.346,-178.510,6.499,148.748
C04337=1172.940,144.090,-55.367,-178.508,6.501,148.748
C04338=1172.935,144.339,-55.387,-178.505,6.502,148.748
C04339=1172.930,144.588,-55.408,-178.502,6.504,148.747
C04340=1172.925,144.837,-55.428,-178.500,6.505,148.747
C04341=1172.920,145.086,-55.449,-178.498,6.507,148.746
C04342=1172.916,145.335,-55.470,-178.495,6.509,148.746
C04343=1172.911,145.584,-55.491,-178.492,6.510,148.746
C04344=1172.907,145.833,-55.512,-178.489,6.512,148.745
C04345=1172.902,146.083,-55.533,-178.486,6.514,148.745
C04346=1172.898,146.332,-55.553,-178.484,6.515,148.744
C04347=1172.892,146.581,-55.574,-178.481,6.517,148.744
C04348=1172.888,146.830,-55.595,-178.478,6.519,148.744
C04349=1172.883,147.079,-55.616,-178.475,6.521,148.743
C04350=1172.879,147.327,-55.637,-178.473,6.522,148.743
C04351=1172.873,147.577,-55.658,-178.470,6.524,148.742
C04352=1172.869,147.826,-55.678,-178.467,6.526,148.742
C04353=1172.864,148.075,-55.699,-178.465,6.528,148.742
C04354=1172.859,148.324,-55.721,-178.462,6.529,148.741
C04355=1172.855,148.573,-55.742,-178.459,6.531,148.741
C04356=1172.850,148.823,-55.763,-178.457,6.532,148.740
C04357=1172.846,149.071,-55.783,-178.455,6.534,148.740
C04358=1172.841,149.320,-55.805,-178.452,6.535,148.740
C04359=1172.835,149.569,-55.826,-178.449,6.537,148.739
C04360=1172.831,149.818,-55.846,-178.446,6.539,148.739
C04361=1172.826,150.067,-55.868,-178.443,6.540,148.738
C04362=1172.822,150.317,-55.889,-178.441,6.542,148.738
C04363=1172.817,150.566,-55.909,-178.438,6.544,148.738
C04364=1172.812,150.814,-55.931,-178.435,6.546,148.737
C04365=1172.807,151.064,-55.952,-178.432,6.547,148.737
C04366=1172.803,151.313,-55.972,-178.430,6.549,148.736
C04367=1172.798,151.562,-55.994,-178.427,6.551,148.736
C04368=1172.793,151.811,-56.015,-178.424,6.553,148.736
C04369=1172.789,152.060,-56.036,-178.422,6.554,148.735
C04370=1172.784,152.309,-56.057,-178.419,6.556,148.735
C04371=1172.779,152.558,-56.078,-178.416,6.558,148.735
C04372=1172.774,152.808,-56.100,-178.414,6.560,148.734
C04373=1172.770,153.056,-56.121,-178.411,6.561,148.734
C04374=1172.765,153.305,-56.142,-178.408,6.563,148.733
C04375=1172.760,153.554,-56.163,-178.406,6.565,148.733
C04376=1172.755,153.804,-56.184,-178.403,6.567,148.733
C04377=1172.751,154.053,-56.206,-178.400,6.568,148.732
C04378=1172.746,154.302,-56.227,-178.397,6.570,148.732
C04379=1172.741,154.551,-56.249,-178.395,6.572,148.732
C04380=1172.736,154.800,-56.269,-178.392,6.574,148.731
C04381=1172.733,155.049,-56.291,-178.389,6.575,148.731
C04382=1172.727,155.298,-56.312,-178.387,6.577,148.730
C04383=1172.723,155.547,-56.334,-178.384,6.579,148.730
C04384=1172.718,155.795,-56.355,-178.381,6.581,148.730
C04385=1172.713,156.045,-56.377,-178.379,6.582,148.729
C04386=1172.708,156.294,-56.398,-178.376,6.584,148.729
C04387=1172.704,156.543,-56.419,-178.373,6.586,148.728
C04388=1172.699,156.792,-56.440,-178.371,6.588,148.728
C04389=1172.695,157.041,-56.462,-178.368,6.589,148.728
C04390=1172.689,157.290,-56.483,-178.365,6.591,148.727
C04391=1172.685,157.539,-56.505,-178.362,6.593,148.727
C04392=1172.680,157.789,-56.526,-178.360,6.595,148.727
C04393=1172.676,158.057,-56.550,-178.357,6.596,148.726
C04394=1172.670,158.327,-56.573,-178.354,6.598,148.726
C04395=1172.665,158.595,-56.596,-178.351,6.600,148.725
C04396=1172.660,158.864,-56.620,-178.348,6.602,148.725
C04397=1172.655,159.114,-56.641,-178.345,6.604,148.725
C04398=1172.650,159.362,-56.663,-178.343,6.606,148.724
C04399=1172.646,159.611,-56.684,-178.340,6.607,148.724
C04400=1172.642,159.860,-56.706,-178.337,6.609,148.723
C04401=1172.637,160.109,-56.727,-178.335,6.611,148.723
C04402=1172.632,160.358,-56.748,-178.332,6.613,148.723
C04403=1172.627,160.607,-56.771,-178.329,6.614,148.722
C04404=1172.623,160.856,-56.792,-178.326,6.616,148.722
C04405=1172.618,161.106,-56.814,-178.324,6.618,148.722
C04406=1172.613,161.354,-56.835,-178.321,6.620,148.721
C04407=1172.608,161.603,-56.857,-178.318,6.622,148.721
C04408=1172.604,161.852,-56.879,-178.316,6.623,148.720
C04409=1172.599,162.101,-56.901,-178.313,6.625,148.720
C04410=1172.594,162.350,-56.922,-178.310,6.627,148.720
C04411=1172.590,162.600,-56.944,-178.308,6.629,148.719
C04412=1172.585,162.848,-56.965,-178.305,6.630,148.719
C04413=1172.580,163.098,-56.987,-178.302,6.633,148.719
C04414=1172.576,163.346,-57.009,-178.299,6.635,148.718
C04415=1172.571,163.596,-57.031,-178.296,6.636,148.718
C04416=1172.566,163.844,-57.053,-178.294,6.639,148.718
C04417=1172.562,164.093,-57.074,-178.291,6.640,148.717
C04418=1172.557,164.342,-57.097,-178.289,6.642,148.717
C04419=1172.552,164.591,-57.118,-178.286,6.644,148.717
C04420=1172.547,164.840,-57.141,-178.283,6.646,148.716
C04421=1172.543,165.089,-57.163,-178.281,6.647,148.716
C04422=1172.538,165.338,-57.185,-178.278,6.649,148.715
C04423=1172.533,165.587,-57.206,-178.275,6.651,148.715
C04424=1172.529,165.836,-57.228,-178.273,6.653,148.715
C04425=1172.524,166.085,-57.250,-178.270,6.654,148.714
C04426=1172.520,166.334,-57.272,-178.267,6.656,148.714
C04427=1172.515,166.583,-57.294,-178.265,6.658,148.714
C04428=1172.510,166.832,-57.315,-178.261,6.660,148.713
C04429=1172.505,167.081,-57.338,-178.259,6.662,148.713
C04430=1172.500,167.330,-57.360,-178.256,6.664,148.713
C04431=1172.496,167.579,-57.382,-178.253,6.666,148.712
C04432=1172.491,167.828,-57.403,-178.251,6.667,148.712
C04433=1172.487,168.077,-57.425,-178.248,6.670,148.712
C04434=1172.481,168.326,-57.448,-178.246,6.671,148.711
C04435=1172.477,168.575,-57.471,-178.243,6.673,148.711
C04436=1172.473,168.824,-57.492,-178.240,6.675,148.711
C04437=1172.468,169.073,-57.514,-178.238,6.677,148.710
C04438=1172.463,169.322,-57.536,-178.235,6.678,148.710
C04439=1172.458,169.571,-57.559,-178.232,6.680,148.709
C04440=1172.454,169.821,-57.581,-178.229,6.683,148.709
C04441=1172.450,170.069,-57.603,-178.226,6.685,148.709
C04442=1172.445,170.318,-57.625,-178.224,6.686,148.708
C04443=1172.440,170.567,-57.647,-178.221,6.688,148.708
C04444=1172.435,170.816,-57.669,-178.218,6.690,148.708
C04445=1172.431,171.065,-57.691,-178.216,6.692,148.707
C04446=1172.426,171.314,-57.714,-178.213,6.694,148.707
C04447=1172.421,171.563,-57.736,-178.211,6.695,148.707
C04448=1172.417,171.812,-57.758,-178.208,6.697,148.706
C04449=1172.413,172.061,-57.781,-178.205,6.700,148.706
C04450=1172.407,172.310,-57.803,-178.202,6.702,148.706
C04451=1172.403,172.559,-57.825,-178.199,6.703,148.705
C04452=1172.398,172.807,-57.848,-178.197,6.705,148.705
C04453=1172.393,173.057,-57.870,-178.194,6.707,148.705
C04454=1172.389,173.306,-57.892,-178.191,6.709,148.704
C04455=1172.385,173.554,-57.915,-178.189,6.711,148.704
C04456=1172.380,173.804,-57.937,-178.186,6.712,148.704
C04457=1172.375,174.052,-57.959,-178.183,6.715,148.703
C04458=1172.370,174.301,-57.982,-178.180,6.717,148.703
C04459=1172.366,174.551,-58.004,-178.178,6.719,148.703
C04460=1172.361,174.799,-58.027,-178.175,6.720,148.702
C04461=1172.356,175.048,-58.050,-178.172,6.722,148.702
C04462=1172.352,175.298,-58.072,-178.170,6.724,148.702
C04463=1172.347,175.546,-58.095,-178.168,6.726,148.701
C04464=1172.342,175.795,-58.117,-178.164,6.729,148.701
C04465=1172.338,176.044,-58.139,-178.162,6.730,148.701
C04466=1172.333,176.293,-58.162,-178.159,6.732,148.700
C04467=1172.329,176.542,-58.184,-178.156,6.734,148.700
C04468=1172.324,176.791,-58.207,-178.154,6.736,148.700
C04469=1172.319,177.039,-58.229,-178.151,6.737,148.699
C04470=1172.314,177.289,-58.252,-178.149,6.740,148.699
C04471=1172.310,177.538,-58.275,-178.145,6.742,148.699
C04472=1172.305,177.787,-58.297,-178.143,6.744,148.698
C04473=1172.301,178.035,-58.320,-178.140,6.746,148.698
C04474=1172.296,178.284,-58.343,-178.137,6.747,148.698
C04475=1172.291,178.533,-58.365,-178.135,6.749,148.697
C04476=1172.286,178.782,-58.388,-178.132,6.751,148.697
C04477=1172.282,179.031,-58.410,-178.129,6.754,148.697
C04478=1172.277,179.281,-58.434,-178.127,6.756,148.696
C04479=1172.273,179.529,-58.456,-178.124,6.757,148.696
C04480=1172.268,179.778,-58.479,-178.121,6.759,148.696
C04481=1172.264,180.027,-58.502,-178.119,6.761,148.695
C04482=1172.259,180.276,-58.525,-178.116,6.763,148.695
C04483=1172.254,180.525,-58.547,-178.113,6.766,148.695
C04484=1172.250,180.774,-58.570,-178.110,6.767,148.695
C04485=1172.245,181.023,-58.593,-178.108,6.769,148.694
C04486=1172.241,181.272,-58.615,-178.105,6.771,148.694
C04487=1172.235,181.520,-58.638,-178.102,6.773,148.693
C04488=1172.231,181.769,-58.661,-178.100,6.775,148.693
C04489=1172.227,182.018,-58.684,-178.097,6.777,148.693
C04490=1172.222,182.268,-58.707,-178.094,6.779,148.693
C04491=1172.217,182.516,-58.729,-178.092,6.781,148.692
C04492=1172.212,182.765,-58.753,-178.089,6.783,148.692
C04493=1172.208,183.013,-58.776,-178.086,6.785,148.692
C04494=1172.204,183.263,-58.799,-178.083,6.787,148.691
C04495=1172.199,183.512,-58.822,-178.081,6.789,148.691
C04496=1172.194,183.760,-58.844,-178.078,6.791,148.691
C04497=1172.189,184.031,-58.869,-178.075,6.793,148.690
C04498=1172.184,184.300,-58.894,-178.072,6.795,148.690
C04499=1172.180,184.569,-58.920,-178.069,6.797,148.690
C04500=1172.175,184.839,-58.945,-178.066,6.800,148.689
C04501=1172.169,185.087,-58.968,-178.063,6.802,148.689
C04502=1172.165,185.336,-58.990,-178.061,6.803,148.689
C04503=1172.160,185.586,-59.013,-178.059,6.805,148.689
C04504=1172.156,185.835,-59.036,-178.055,6.808,148.688
C04505=1172.151,186.084,-59.060,-178.053,6.810,148.688
C04506=1172.147,186.333,-59.083,-178.050,6.812,148.687
C04507=1172.142,186.582,-59.106,-178.048,6.814,148.687
C04508=1172.137,186.830,-59.129,-178.045,6.816,148.687
C04509=1172.132,187.079,-59.152,-178.042,6.818,148.687
C04510=1172.128,187.328,-59.175,-178.039,6.820,148.686
C04511=1172.124,187.577,-59.198,-178.037,6.822,148.686
C04512=1172.119,187.826,-59.222,-178.034,6.824,148.686
C04513=1172.114,188.075,-59.245,-178.031,6.826,148.685
C04514=1172.109,188.324,-59.268,-178.028,6.828,148.685
C04515=1172.106,188.572,-59.291,-178.026,6.830,148.685
C04516=1172.101,188.822,-59.315,-178.024,6.832,148.685
C04517=1172.096,189.069,-59.338,-178.020,6.835,148.684
C04518=1172.091,189.318,-59.362,-178.018,6.836,148.684
C04519=1172.086,189.567,-59.385,-178.015,6.838,148.684
C04520=1172.082,189.816,-59.408,-178.012,6.840,148.683
C04521=1172.077,190.065,-59.432,-178.009,6.843,148.683
C04522=1172.073,190.314,-59.454,-178.007,6.845,148.683
C04523=1172.068,190.563,-59.478,-178.004,6.846,148.682
C04524=1172.064,190.812,-59.501,-178.001,6.848,148.682
C04525=1172.059,191.061,-59.525,-177.999,6.851,148.682
C04526=1172.055,191.310,-59.549,-177.996,6.853,148.682
C04527=1172.050,191.559,-59.572,-177.993,6.855,148.681
C04528=1172.045,191.808,-59.595,-177.991,6.856,148.681
C04529=1172.040,192.057,-59.619,-177.988,6.859,148.681
C04530=1172.036,192.305,-59.643,-177.985,6.861,148.680
C04531=1172.031,192.554,-59.666,-177.983,6.863,148.680
C04532=1172.027,192.803,-59.689,-177.980,6.865,148.680
C04533=1172.022,193.052,-59.713,-177.977,6.868,148.680
C04534=1172.018,193.301,-59.737,-177.974,6.869,148.679
C04535=1172.013,193.550,-59.760,-177.972,6.871,148.679
C04536=1172.008,193.799,-59.784,-177.970,6.873,148.679
C04537=1172.005,194.047,-59.807,-177.966,6.876,148.678
C04538=1172.000,194.296,-59.830,-177.964,6.878,148.678
C04539=1171.994,194.545,-59.854,-177.961,6.879,148.678
C04540=1171.990,194.794,-59.879,-177.958,6.882,148.678
C04541=1171.985,195.043,-59.902,-177.955,6.884,148.677
C04542=1171.981,195.292,-59.925,-177.953,6.886,148.677
C04543=1171.976,195.540,-59.949,-177.950,6.888,148.677
C04544=1171.971,195.789,-59.973,-177.947,6.891,148.676
C04545=1171.967,196.038,-59.996,-177.945,6.892,148.676
C04546=1171.962,196.287,-60.020,-177.942,6.894,148.676
C04547=1171.958,196.536,-60.043,-177.939,6.897,148.676
C04548=1171.953,196.784,-60.068,-177.937,6.899,148.675
C04549=1171.949,197.033,-60.091,-177.934,6.901,148.675
C04550=1171.944,197.281,-60.115,-177.932,6.903,148.675
C04551=1171.940,197.530,-60.138,-177.928,6.905,148.675
C04552=1171.935,197.779,-60.162,-177.926,6.907,148.674
C04553=1171.931,198.029,-60.186,-177.923,6.909,148.674
C04554=1171.926,198.277,-60.211,-177.920,6.912,148.674
C04555=1171.921,198.526,-60.234,-177.918,6.914,148.673
C04556=1171.917,198.775,-60.258,-177.915,6.915,148.673
C04557=1171.912,199.024,-60.282,-177.912,6.918,148.673
C04558=1171.908,199.272,-60.306,-177.910,6.920,148.673
C04559=1171.903,199.521,-60.329,-177.907,6.922,148.672
C04560=1171.899,199.770,-60.353,-177.905,6.924,148.672
C04561=1171.893,200.018,-60.378,-177.901,6.927,148.672
C04562=1171.889,200.268,-60.401,-177.899,6.928,148.671
C04563=1171.885,200.517,-60.426,-177.897,6.931,148.671
C04564=1171.880,200.766,-60.449,-177.893,6.933,148.671
C04565=1171.876,201.014,-60.473,-177.891,6.935,148.671
C04566=1171.871,201.263,-60.498,-177.888,6.937,148.671
C04567=1171.866,201.512,-60.521,-177.885,6.940,148.670
C04568=1171.862,201.761,-60.545,-177.883,6.941,148.670
C04569=1171.858,202.009,-60.570,-177.880,6.944,148.670
C04570=1171.852,202.259,-60.593,-177.877,6.946,148.669
C04571=1171.848,202.507,-60.618,-177.874,6.948,148.669
C04572=1171.844,202.755,-60.642,-177.872,6.950,148.669
C04573=1171.839,203.004,-60.666,-177.869,6.953,148.669
C04574=1171.834,203.254,-60.690,-177.866,6.955,148.668
C04575=1171.830,203.502,-60.714,-177.864,6.957,148.668
C04576=1171.826,203.751,-60.738,-177.861,6.959,148.668
C04577=1171.821,203.999,-60.762,-177.858,6.961,148.667
C04578=1171.817,204.249,-60.787,-177.856,6.963,148.667
C04579=1171.812,204.498,-60.811,-177.853,6.966,148.667
C04580=1171.808,204.746,-60.835,-177.850,6.968,148.667
C04581=1171.802,204.995,-60.859,-177.848,6.970,148.667
C04582=1171.798,205.243,-60.883,-177.845,6.972,148.666
C04583=1171.794,205.492,-60.908,-177.842,6.974,148.666
C04584=1171.789,205.741,-60.933,-177.839,6.977,148.666
C04585=1171.784,205.990,-60.956,-177.837,6.979,148.665
C04586=1171.779,206.239,-60.981,-177.834,6.981,148.665
C04587=1171.776,206.488,-61.005,-177.831,6.983,148.665
C04588=1171.771,206.736,-61.029,-177.829,6.985,148.665
C04589=1171.766,206.985,-61.054,-177.826,6.987,148.665
C04590=1171.762,207.233,-61.078,-177.823,6.990,148.664
C04591=1171.757,207.483,-61.103,-177.820,6.992,148.664
C04592=1171.753,207.731,-61.127,-177.818,6.994,148.664
C04593=1171.748,207.980,-61.151,-177.815,6.997,148.663
C04594=1171.744,208.229,-61.176,-177.813,6.999,148.663
C04595=1171.739,208.477,-61.200,-177.810,7.001,148.663
C04596=1171.734,208.726,-61.225,-177.807,7.003,148.663
C04597=1171.730,208.975,-61.249,-177.805,7.005,148.663
C04598=1171.725,209.224,-61.274,-177.801,7.008,148.662
C04599=1171.721,209.472,-61.298,-177.799,7.010,148.662
C04600=1171.716,209.721,-61.323,-177.797,7.012,148.662
C04601=1171.711,209.992,-61.350,-177.793,7.014,148.661
C04602=1171.706,210.262,-61.376,-177.790,7.017,148.661
C04603=1171.701,210.532,-61.403,-177.788,7.019,148.661
C04604=1171.696,210.803,-61.430,-177.785,7.022,148.661
C04605=1171.692,211.052,-61.454,-177.781,7.024,148.660
C04606=1171.687,211.301,-61.479,-177.779,7.026,148.660
C04607=1171.683,211.549,-61.503,-177.777,7.028,148.660
C04608=1171.678,211.798,-61.528,-177.774,7.031,148.660
C04609=1171.674,212.047,-61.553,-177.771,7.033,148.660
C04610=1171.669,212.295,-61.578,-177.768,7.035,148.659
C04611=1171.665,212.544,-61.602,-177.766,7.038,148.659
C04612=1171.660,212.793,-61.627,-177.763,7.039,148.659
C04613=1171.655,213.042,-61.652,-177.760,7.042,148.659
C04614=1171.651,213.291,-61.676,-177.758,7.044,148.658
C04615=1171.647,213.539,-61.702,-177.755,7.047,148.658
C04616=1171.642,213.788,-61.726,-177.752,7.049,148.658
C04617=1171.638,214.037,-61.751,-177.750,7.051,148.658
C04618=1171.633,214.286,-61.775,-177.747,7.054,148.657
C04619=1171.629,214.534,-61.800,-177.744,7.055,148.657
C04620=1171.624,214.783,-61.825,-177.741,7.058,148.657
C04621=1171.619,215.032,-61.850,-177.739,7.060,148.657
C04622=1171.615,215.280,-61.875,-177.736,7.063,148.657
C04623=1171.610,215.529,-61.900,-177.733,7.065,148.656
C04624=1171.606,215.778,-61.925,-177.731,7.067,148.656
C04625=1171.602,216.026,-61.949,-177.728,7.070,148.656
C04626=1171.597,216.276,-61.975,-177.725,7.071,148.655
C04627=1171.592,216.524,-62.000,-177.722,7.074,148.655
C04628=1171.588,216.773,-62.025,-177.720,7.076,148.655
C04629=1171.583,217.022,-62.049,-177.717,7.079,148.655
C04630=1171.579,217.270,-62.075,-177.714,7.081,148.655
C04631=1171.574,217.519,-62.099,-177.712,7.083,148.655
C04632=1171.570,217.768,-62.125,-177.709,7.086,148.654
C04633=1171.565,218.016,-62.149,-177.707,7.088,148.654
C04634=1171.561,218.265,-62.175,-177.703,7.090,148.654
C04635=1171.556,218.514,-62.200,-177.701,7.092,148.654
C04636=1171.552,218.762,-62.225,-177.698,7.095,148.653
C04637=1171.547,219.011,-62.249,-177.696,7.097,148.653
C04638=1171.543,219.260,-62.275,-177.693,7.100,148.653
C04639=1171.538,219.509,-62.300,-177.690,7.102,148.653
C04640=1171.534,219.757,-62.326,-177.688,7.104,148.652
C04641=1171.529,220.006,-62.350,-177.684,7.106,148.652
C04642=1171.525,220.255,-62.375,-177.682,7.109,148.652
C04643=1171.520,220.503,-62.400,-177.679,7.111,148.652
C04644=1171.516,220.752,-62.426,-177.677,7.113,148.652
C04645=1171.511,221.000,-62.451,-177.674,7.116,148.651
C04646=1171.506,221.250,-62.476,-177.671,7.118,148.651
C04647=1171.502,221.498,-62.502,-177.668,7.121,148.651
C04648=1171.498,221.746,-62.527,-177.666,7.123,148.651
C04649=1171.494,221.996,-62.552,-177.663,7.125,148.651
C04650=1171.489,222.244,-62.577,-177.661,7.127,148.650
C04651=1171.485,222.493,-62.603,-177.657,7.130,148.650
C04652=1171.479,222.741,-62.628,-177.655,7.132,148.650
C04653=1171.475,222.990,-62.653,-177.652,7.135,148.650
C04654=1171.471,223.239,-62.679,-177.650,7.137,148.650
C04655=1171.466,223.487,-62.705,-177.647,7.140,148.649
C04656=1171.462,223.736,-62.730,-177.644,7.142,148.649
C04657=1171.457,223.984,-62.755,-177.642,7.145,148.649
C04658=1171.453,224.233,-62.781,-177.639,7.146,148.649
C04659=1171.448,224.482,-62.807,-177.636,7.149,148.649
C04660=1171.443,224.731,-62.831,-177.634,7.151,148.648
C04661=1171.439,224.980,-62.857,-177.631,7.153,148.648
C04662=1171.434,225.228,-62.882,-177.628,7.156,148.648
C04663=1171.430,225.477,-62.908,-177.626,7.158,148.648
C04664=1171.426,225.725,-62.934,-177.623,7.161,148.647
C04665=1171.421,225.973,-62.959,-177.620,7.163,148.647
C04666=1171.416,226.223,-62.984,-177.617,7.165,148.647
C04667=1171.412,226.472,-63.010,-177.614,7.168,148.647
C04668=1171.407,226.720,-63.035,-177.612,7.170,148.647
C04669=1171.403,226.969,-63.061,-177.609,7.173,148.647
C04670=1171.399,227.217,-63.087,-177.607,7.175,148.646
C04671=1171.394,227.465,-63.112,-177.604,7.178,148.646
C04672=1171.390,227.714,-63.138,-177.601,7.180,148.646
C04673=1171.386,227.963,-63.164,-177.598,7.183,148.646
C04674=1171.381,228.212,-63.190,-177.596,7.185,148.646
C04675=1171.377,228.460,-63.215,-177.593,7.187,148.645
C04676=1171.372,228.709,-63.241,-177.591,7.190,148.645
C04677=1171.368,228.958,-63.266,-177.587,7.192,148.645
C04678=1171.363,229.206,-63.292,-177.585,7.194,148.645
C04679=1171.358,229.455,-63.318,-177.582,7.197,148.645
C04680=1171.354,229.704,-63.344,-177.580,7.199,148.644
C04681=1171.350,229.952,-63.370,-177.577,7.202,148.644
C04682=1171.345,230.201,-63.395,-177.574,7.204,148.644
C04683=1171.341,230.449,-63.421,-177.572,7.207,148.644
C04684=1171.337,230.698,-63.447,-177.569,7.209,148.644
C04685=1171.332,230.947,-63.473,-177.566,7.211,148.644
C04686=1171.327,231.195,-63.498,-177.563,7.214,148.643
C04687=1171.323,231.444,-63.525,-177.561,7.216,148.643
C04688=1171.319,231.692,-63.550,-177.558,7.219,148.643
C04689=1171.314,231.941,-63.576,-177.555,7.221,148.643
C04690=1171.309,232.190,-63.602,-177.553,7.224,148.643
C04691=1171.305,232.438,-63.628,-177.550,7.226,148.643
C04692=1171.300,232.687,-63.654,-177.547,7.229,148.642
C04693=1171.296,232.935,-63.680,-177.545,7.231,148.642
C04694=1171.291,233.184,-63.706,-177.542,7.234,148.642
C04695=1171.287,233.433,-63.732,-177.540,7.236,148.642
C04696=1171.282,233.681,-63.758,-177.537,7.239,148.642
C04697=1171.278,233.930,-63.783,-177.534,7.241,148.641
C04698=1171.274,234.179,-63.810,-177.531,7.243,148.641
C04699=1171.269,234.428,-63.836,-177.529,7.246,148.641
C04700=1171.265,234.676,-63.862,-177.526,7.248,148.641
C04701=1171.260,234.924,-63.889,-177.523,7.251,148.641
C04702=1171.256,235.173,-63.914,-177.521,7.253,148.641
C04703=1171.251,235.422,-63.940,-177.518,7.256,148.640
C04704=1171.247,235.670,-63.967,-177.515,7.259,148.640
C04705=1171.242,235.942,-63.995,-177.512,7.261,148.640
C04706=1171.238,236.213,-64.024,-177.510,7.263,148.640
C04707=1171.232,236.485,-64.052,-177.506,7.266,148.640
C04708=1171.227,236.756,-64.081,-177.504,7.269,148.640
C04709=1171.223,237.005,-64.107,-177.501,7.272,148.639
C04710=1171.218,237.253,-64.134,-177.498,7.274,148.639
C04711=1171.214,237.502,-64.160,-177.496,7.277,148.639
C04712=1171.209,237.751,-64.186,-177.493,7.280,148.639
C04713=1171.205,238.000,-64.212,-177.490,7.282,148.639
C04714=1171.201,238.248,-64.238,-177.487,7.284,148.639
C04715=1171.196,238.497,-64.265,-177.485,7.287,148.639
C04716=1171.192,238.746,-64.291,-177.482,7.289,148.638
C04717=1171.187,238.993,-64.318,-177.479,7.292,148.638
C04718=1171.183,239.242,-64.343,-177.477,7.294,148.638
C04719=1171.178,239.491,-64.370,-177.474,7.297,148.638
C04720=1171.174,239.740,-64.396,-177.472,7.299,148.638
C04721=1171.169,239.988,-64.423,-177.469,7.302,148.638
C04722=1171.165,240.236,-64.450,-177.466,7.305,148.637
C04723=1171.160,240.485,-64.476,-177.463,7.307,148.637
C04724=1171.156,240.734,-64.503,-177.461,7.310,148.637
C04725=1171.151,240.983,-64.529,-177.458,7.312,148.637
C04726=1171.147,241.231,-64.555,-177.455,7.315,148.637
C04727=1171.143,241.479,-64.582,-177.453,7.317,148.637
C04728=1171.139,241.728,-64.608,-177.450,7.319,148.636
C04729=1171.134,241.977,-64.635,-177.447,7.322,148.636
C04730=1171.130,242.225,-64.662,-177.444,7.325,148.636
C04731=1171.125,242.474,-64.688,-177.442,7.327,148.636
C04732=1171.121,242.722,-64.715,-177.439,7.330,148.636
C04733=1171.116,242.971,-64.742,-177.437,7.332,148.636
C04734=1171.112,243.220,-64.768,-177.434,7.335,148.636
C04735=1171.108,243.468,-64.794,-177.431,7.338,148.635
C04736=1171.103,243.716,-64.821,-177.429,7.340,148.635
C04737=1171.099,243.965,-64.848,-177.426,7.343,148.635
C04738=1171.094,244.214,-64.874,-177.423,7.346,148.635
C04739=1171.089,244.462,-64.901,-177.420,7.348,148.635
C04740=1171.085,244.710,-64.928,-177.418,7.351,148.635
C04741=1171.081,244.959,-64.955,-177.415,7.353,148.635
C04742=1171.076,245.207,-64.982,-177.413,7.356,148.635
C04743=1171.072,245.456,-65.008,-177.410,7.358,148.634
C04744=1171.067,245.705,-65.035,-177.407,7.360,148.634
C04745=1171.063,245.953,-65.062,-177.405,7.363,148.634
C04746=1171.059,246.201,-65.088,-177.402,7.366,148.634
C04747=1171.054,246.450,-65.115,-177.399,7.368,148.634
C04748=1171.049,246.698,-65.142,-177.396,7.371,148.634
C04749=1171.045,246.947,-65.169,-177.394,7.374,148.634
C04750=1171.041,247.196,-65.196,-177.392,7.376,148.634
C04751=1171.037,247.444,-65.223,-177.388,7.379,148.633
C04752=1171.032,247.693,-65.250,-177.386,7.382,148.633
C04753=1171.028,247.941,-65.277,-177.383,7.384,148.633
C04754=1171.023,248.190,-65.303,-177.381,7.387,148.633
C04755=1171.019,248.439,-65.330,-177.378,7.390,148.633
C04756=1171.014,248.687,-65.357,-177.375,7.392,148.633
C04757=1171.010,248.935,-65.384,-177.372,7.395,148.633
C04758=1171.006,249.183,-65.412,-177.370,7.398,148.632
C04759=1171.002,249.432,-65.439,-177.368,7.400,148.632
C04760=1170.997,249.681,-65.466,-177.364,7.402,148.632
C04761=1170.992,249.929,-65.493,-177.362,7.405,148.632
C04762=1170.988,250.177,-65.520,-177.359,7.407,148.632
C04763=1170.984,250.426,-65.547,-177.357,7.410,148.632
C04764=1170.979,250.674,-65.574,-177.354,7.413,148.632
C04765=1170.974,250.923,-65.601,-177.351,7.415,148.632
C04766=1170.970,251.172,-65.628,-177.348,7.418,148.631
C04767=1170.966,251.421,-65.655,-177.346,7.421,148.631
C04768=1170.962,251.669,-65.682,-177.343,7.424,148.631
C04769=1170.957,251.917,-65.710,-177.341,7.426,148.631
C04770=1170.953,252.165,-65.737,-177.338,7.429,148.631
C04771=1170.948,252.414,-65.764,-177.335,7.432,148.631
C04772=1170.944,252.663,-65.791,-177.333,7.434,148.631
C04773=1170.939,252.911,-65.818,-177.330,7.437,148.631
C04774=1170.935,253.159,-65.846,-177.327,7.440,148.631
C04775=1170.930,253.408,-65.873,-177.325,7.442,148.631
C04776=1170.926,253.657,-65.900,-177.322,7.445,148.631
C04777=1170.922,253.905,-65.927,-177.319,7.448,148.630
C04778=1170.917,254.153,-65.955,-177.316,7.451,148.630
C04779=1170.913,254.402,-65.982,-177.314,7.453,148.630
C04780=1170.909,254.650,-66.009,-177.311,7.456,148.630
C04781=1170.905,254.899,-66.037,-177.309,7.459,148.630
C04782=1170.900,255.147,-66.064,-177.306,7.461,148.630
C04783=1170.896,255.396,-66.091,-177.303,7.463,148.630
C04784=1170.891,255.643,-66.119,-177.300,7.466,148.630
C04785=1170.887,255.893,-66.146,-177.298,7.469,148.629
C04786=1170.883,256.141,-66.173,-177.295,7.471,148.629
C04787=1170.878,256.389,-66.201,-177.293,7.474,148.629
C04788=1170.873,256.639,-66.229,-177.290,7.477,148.629
C04789=1170.869,256.886,-66.257,-177.288,7.479,148.629
C04790=1170.864,257.135,-66.284,-177.285,7.482,148.629
C04791=1170.860,257.383,-66.312,-177.282,7.485,148.629
C04792=1170.856,257.632,-66.339,-177.279,7.488,148.629
C04793=1170.851,257.881,-66.366,-177.277,7.490,148.629
C04794=1170.847,258.128,-66.394,-177.274,7.493,148.629
C04795=1170.843,258.378,-66.421,-177.271,7.496,148.629
C04796=1170.839,258.625,-66.449,-177.269,7.499,148.629
C04797=1170.834,258.874,-66.476,-177.266,7.501,148.628
C04798=1170.830,259.123,-66.504,-177.264,7.504,148.628
C04799=1170.826,259.370,-66.532,-177.260,7.507,148.628
C04800=1170.820,259.619,-66.560,-177.258,7.509,148.628
C04801=1170.817,259.868,-66.588,-177.256,7.512,148.628
C04802=1170.812,260.116,-66.615,-177.253,7.515,148.628
C04803=1170.808,260.364,-66.643,-177.250,7.518,148.628
C04804=1170.804,260.613,-66.671,-177.248,7.520,148.628
C04805=1170.799,260.861,-66.698,-177.245,7.523,148.628
C04806=1170.794,261.109,-66.726,-177.242,7.526,148.628
C04807=1170.790,261.359,-66.754,-177.240,7.529,148.628
C04808=1170.786,261.606,-66.782,-177.237,7.531,148.627
C04809=1170.781,261.880,-66.812,-177.234,7.535,148.627
C04810=1170.776,262.153,-66.843,-177.231,7.537,148.627
C04811=1170.771,262.426,-66.873,-177.228,7.540,148.627
C04812=1170.767,262.699,-66.904,-177.225,7.543,148.627
C04813=1170.762,262.947,-66.932,-177.223,7.546,148.627
C04814=1170.758,263.196,-66.960,-177.220,7.549,148.627
C04815=1170.753,263.444,-66.988,-177.218,7.551,148.627
C04816=1170.749,263.693,-67.016,-177.215,7.554,148.627
C04817=1170.745,263.941,-67.043,-177.212,7.557,148.627
C04818=1170.741,264.189,-67.072,-177.209,7.560,148.627
C04819=1170.736,264.438,-67.100,-177.207,7.563,148.627
C04820=1170.732,264.685,-67.128,-177.205,7.565,148.627
C04821=1170.728,264.935,-67.155,-177.202,7.568,148.627
C04822=1170.723,265.183,-67.184,-177.199,7.571,148.626
C04823=1170.719,265.431,-67.212,-177.196,7.574,148.626
C04824=1170.715,265.679,-67.239,-177.194,7.576,148.626
C04825=1170.710,265.928,-67.268,-177.191,7.579,148.626
C04826=1170.706,266.176,-67.296,-177.188,7.582,148.626
C04827=1170.701,266.425,-67.325,-177.185,7.585,148.626
C04828=1170.697,266.673,-67.352,-177.183,7.587,148.626
C04829=1170.693,266.921,-67.381,-177.181,7.590,148.626
C04830=1170.688,267.170,-67.409,-177.178,7.593,148.626
C04831=1170.684,267.419,-67.436,-177.175,7.596,148.626
C04832=1170.680,267.667,-67.464,-177.172,7.599,148.626
C04833=1170.675,267.916,-67.493,-177.170,7.601,148.626
C04834=1170.671,268.163,-67.521,-177.167,7.604,148.626
C04835=1170.666,268.412,-67.549,-177.165,7.607,148.625
C04836=1170.662,268.660,-67.578,-177.162,7.610,148.625
C04837=1170.658,268.908,-67.607,-177.159,7.613,148.625
C04838=1170.653,269.156,-67.634,-177.157,7.615,148.625
C04839=1170.649,269.405,-67.663,-177.154,7.618,148.625
C04840=1170.645,269.653,-67.691,-177.151,7.621,148.625
C04841=1170.640,269.902,-67.720,-177.149,7.624,148.625
C04842=1170.636,270.150,-67.747,-177.146,7.627,148.625
C04843=1170.631,270.399,-67.776,-177.144,7.629,148.625
C04844=1170.627,270.647,-67.804,-177.141,7.632,148.625
C04845=1170.622,270.895,-67.833,-177.138,7.635,148.625
C04846=1170.619,271.143,-67.862,-177.136,7.638,148.625
C04847=1170.614,271.392,-67.890,-177.133,7.641,148.625
C04848=1170.610,271.640,-67.918,-177.130,7.644,148.625
C04849=1170.606,271.889,-67.947,-177.128,7.646,148.625
C04850=1170.601,272.137,-67.975,-177.125,7.649,148.625
C04851=1170.597,272.385,-68.004,-177.123,7.653,148.625
C04852=1170.593,272.633,-68.032,-177.120,7.655,148.625
C04853=1170.588,272.882,-68.061,-177.117,7.658,148.625
C04854=1170.584,273.131,-68.089,-177.115,7.661,148.625
C04855=1170.580,273.378,-68.118,-177.112,7.664,148.625
C04856=1170.575,273.627,-68.147,-177.110,7.667,148.625
C04857=1170.571,273.875,-68.174,-177.107,7.669,148.624
C04858=1170.567,274.123,-68.204,-177.104,7.672,148.624
C04859=1170.562,274.372,-68.233,-177.101,7.675,148.624
C04860=1170.558,274.620,-68.260,-177.099,7.678,148.624
C04861=1170.554,274.868,-68.290,-177.097,7.681,148.624
C04862=1170.549,275.117,-68.318,-177.094,7.684,148.624
C04863=1170.545,275.365,-68.346,-177.091,7.686,148.624
C04864=1170.541,275.613,-68.376,-177.088,7.689,148.624
C04865=1170.536,275.862,-68.404,-177.086,7.692,148.624
C04866=1170.532,276.109,-68.433,-177.083,7.695,148.624
C04867=1170.528,276.358,-68.462,-177.081,7.698,148.624
C04868=1170.523,276.607,-68.490,-177.078,7.701,148.624
C04869=1170.520,276.855,-68.519,-177.076,7.704,148.624
C04870=1170.515,277.103,-68.548,-177.073,7.707,148.624
C04871=1170.510,277.352,-68.577,-177.070,7.710,148.624
C04872=1170.506,277.600,-68.606,-177.067,7.713,148.624
C04873=1170.502,277.848,-68.634,-177.065,7.715,148.624
C04874=1170.497,278.097,-68.663,-177.062,7.718,148.624
C04875=1170.493,278.345,-68.693,-177.060,7.721,148.624
C04876=1170.489,278.593,-68.722,-177.057,7.724,148.624
C04877=1170.485,278.841,-68.750,-177.054,7.727,148.624
C04878=1170.481,279.089,-68.779,-177.052,7.730,148.624
C04879=1170.476,279.338,-68.808,-177.049,7.733,148.624
C04880=1170.472,279.586,-68.837,-177.046,7.736,148.624
C04881=1170.467,279.834,-68.867,-177.044,7.738,148.624
C04882=1170.463,280.083,-68.895,-177.041,7.741,148.624
C04883=1170.459,280.331,-68.924,-177.039,7.744,148.624
C04884=1170.455,280.580,-68.953,-177.036,7.747,148.624
C04885=1170.450,280.828,-68.982,-177.033,7.750,148.624
C04886=1170.446,281.076,-69.011,-177.031,7.753,148.624
C04887=1170.442,281.324,-69.041,-177.028,7.756,148.624
C04888=1170.437,281.573,-69.070,-177.025,7.759,148.624
C04889=1170.433,281.821,-69.099,-177.023,7.761,148.624
C04890=1170.429,282.068,-69.128,-177.021,7.764,148.624
C04891=1170.424,282.317,-69.156,-177.018,7.767,148.623
C04892=1170.420,282.565,-69.186,-177.015,7.770,148.623
C04893=1170.416,282.814,-69.215,-177.012,7.773,148.623
C04894=1170.412,283.062,-69.245,-177.010,7.777,148.624
C04895=1170.408,283.310,-69.274,-177.007,7.780,148.624
C04896=1170.403,283.558,-69.302,-177.005,7.783,148.624
C04897=1170.398,283.807,-69.332,-177.002,7.785,148.623
C04898=1170.394,284.055,-69.361,-177.000,7.788,148.623
C04899=1170.390,284.303,-69.391,-176.997,7.791,148.623
C04900=1170.386,284.551,-69.420,-176.995,7.794,148.624
C04901=1170.382,284.800,-69.450,-176.992,7.797,148.623
C04902=1170.377,285.047,-69.479,-176.989,7.800,148.623
C04903=1170.372,285.296,-69.508,-176.986,7.803,148.623
C04904=1170.368,285.544,-69.537,-176.984,7.806,148.623
C04905=1170.364,285.793,-69.566,-176.981,7.809,148.623
C04906=1170.360,286.041,-69.596,-176.979,7.812,148.624
C04907=1170.356,286.289,-69.625,-176.976,7.814,148.623
C04908=1170.351,286.538,-69.655,-176.974,7.817,148.623
C04909=1170.347,286.786,-69.684,-176.971,7.820,148.623
C04910=1170.343,287.034,-69.714,-176.968,7.823,148.623
C04911=1170.338,287.282,-69.743,-176.966,7.826,148.624
C04912=1170.334,287.530,-69.772,-176.963,7.829,148.623
C04913=1170.329,287.805,-69.806,-176.960,7.832,148.623
C04914=1170.325,288.080,-69.838,-176.957,7.836,148.623
C04915=1170.320,288.355,-69.871,-176.954,7.839,148.623
C04916=1170.316,288.630,-69.903,-176.952,7.842,148.623
C04917=1170.311,288.878,-69.933,-176.949,7.845,148.623
C04918=1170.306,289.126,-69.963,-176.947,7.848,148.624
C04919=1170.302,289.374,-69.993,-176.944,7.851,148.623
C04920=1170.298,289.622,-70.022,-176.941,7.854,148.623
C04921=1170.294,289.870,-70.052,-176.938,7.857,148.623
C04922=1170.290,290.118,-70.081,-176.936,7.861,148.624
C04923=1170.285,290.367,-70.111,-176.933,7.864,148.624
C04924=1170.280,290.615,-70.141,-176.931,7.867,148.624
C04925=1170.277,290.863,-70.171,-176.928,7.870,148.623
C04926=1170.272,291.111,-70.200,-176.925,7.872,148.623
C04927=1170.268,291.359,-70.230,-176.923,7.875,148.624
C04928=1170.264,291.608,-70.259,-176.921,7.878,148.624
C04929=1170.259,291.856,-70.290,-176.918,7.881,148.624
C04930=1170.255,292.104,-70.319,-176.915,7.884,148.624
C04931=1170.251,292.352,-70.349,-176.913,7.887,148.624
C04932=1170.247,292.600,-70.378,-176.910,7.890,148.624
C04933=1170.242,292.848,-70.409,-176.907,7.893,148.624
C04934=1170.238,293.097,-70.439,-176.905,7.896,148.624
C04935=1170.234,293.346,-70.468,-176.902,7.899,148.624
C04936=1170.230,293.594,-70.499,-176.900,7.902,148.624
C04937=1170.226,293.842,-70.529,-176.897,7.905,148.624
C04938=1170.222,294.090,-70.558,-176.894,7.908,148.624
C04939=1170.218,294.338,-70.588,-176.892,7.912,148.624
C04940=1170.213,294.586,-70.618,-176.889,7.915,148.624
C04941=1170.209,294.834,-70.648,-176.886,7.918,148.624
C04942=1170.205,295.082,-70.678,-176.884,7.921,148.624
C04943=1170.200,295.330,-70.709,-176.881,7.924,148.624
C04944=1170.196,295.579,-70.738,-176.879,7.927,148.624
C04945=1170.192,295.826,-70.768,-176.877,7.929,148.624
C04946=1170.187,296.075,-70.798,-176.874,7.932,148.624
C04947=1170.183,296.322,-70.828,-176.871,7.935,148.624
C04948=1170.179,296.572,-70.859,-176.869,7.938,148.624
C04949=1170.175,296.819,-70.889,-176.866,7.942,148.624
C04950=1170.171,297.068,-70.918,-176.864,7.944,148.624
C04951=1170.166,297.316,-70.949,-176.861,7.947,148.624
C04952=1170.162,297.564,-70.979,-176.858,7.950,148.624
C04953=1170.157,297.812,-71.009,-176.856,7.954,148.624
C04954=1170.153,298.060,-71.039,-176.853,7.957,148.624
C04955=1170.149,298.308,-71.070,-176.850,7.960,148.624
C04956=1170.145,298.556,-71.100,-176.848,7.963,148.624
C04957=1170.140,298.805,-71.130,-176.845,7.966,148.624
C04958=1170.137,299.053,-71.160,-176.843,7.969,148.624
C04959=1170.133,299.300,-71.191,-176.840,7.972,148.625
C04960=1170.128,299.549,-71.221,-176.838,7.975,148.624
C04961=1170.124,299.796,-71.251,-176.835,7.978,148.624
C04962=1170.120,300.045,-71.282,-176.833,7.981,148.625
C04963=1170.115,300.294,-71.312,-176.830,7.984,148.625
C04964=1170.111,300.541,-71.342,-176.827,7.987,148.625
C04965=1170.106,300.789,-71.373,-176.825,7.991,148.625
C04966=1170.103,301.037,-71.403,-176.822,7.994,148.625
C04967=1170.098,301.286,-71.434,-176.819,7.997,148.625
C04968=1170.094,301.534,-71.464,-176.817,8.000,148.625
C04969=1170.090,301.782,-71.494,-176.814,8.003,148.625
C04970=1170.086,302.029,-71.525,-176.812,8.006,148.625
C04971=1170.081,302.278,-71.555,-176.809,8.009,148.625
C04972=1170.077,302.527,-71.586,-176.807,8.012,148.625
C04973=1170.073,302.774,-71.616,-176.804,8.015,148.625
C04974=1170.068,303.022,-71.647,-176.802,8.018,148.625
C04975=1170.064,303.270,-71.677,-176.799,8.021,148.625
C04976=1170.061,303.519,-71.708,-176.796,8.024,148.625
C04977=1170.056,303.767,-71.739,-176.794,8.028,148.625
C04978=1170.052,304.014,-71.769,-176.791,8.031,148.625
C04979=1170.047,304.262,-71.800,-176.789,8.034,148.625
C04980=1170.043,304.511,-71.830,-176.786,8.037,148.625
C04981=1170.039,304.759,-71.861,-176.783,8.040,148.625
C04982=1170.035,305.007,-71.891,-176.781,8.043,148.626
C04983=1170.031,305.256,-71.922,-176.778,8.046,148.626
C04984=1170.026,305.504,-71.953,-176.776,8.050,148.626
C04985=1170.022,305.751,-71.983,-176.773,8.052,148.626
C04986=1170.018,305.999,-72.014,-176.771,8.055,148.626
C04987=1170.014,306.248,-72.045,-176.768,8.059,148.626
C04988=1170.009,306.496,-72.076,-176.766,8.062,148.626
C04989=1170.005,306.744,-72.106,-176.763,8.065,148.626
C04990=1170.001,306.992,-72.138,-176.761,8.068,148.626
C04991=1169.997,307.240,-72.169,-176.758,8.071,148.626
C04992=1169.992,307.488,-72.199,-176.756,8.074,148.626
C04993=1169.989,307.736,-72.230,-176.753,8.077,148.626
C04994=1169.984,307.984,-72.261,-176.750,8.081,148.626
C04995=1169.980,308.232,-72.291,-176.748,8.084,148.626
C04996=1169.976,308.480,-72.323,-176.745,8.087,148.626
C04997=1169.971,308.728,-72.353,-176.743,8.090,148.627
C04998=1169.967,308.975,-72.384,-176.740,8.093,148.627
C04999=1169.963,309.224,-72.415,-176.738,8.096,148.627
C05000=1169.959,309.472,-72.446,-176.735,8.099,148.627
C05001=1169.954,309.720,-72.477,-176.733,8.102,148.627
C05002=1169.950,309.969,-72.508,-176.730,8.105,148.627
C05003=1169.946,310.216,-72.539,-176.727,8.108,148.627
C05004=1169.942,310.465,-72.571,-176.725,8.112,148.627
C05005=1169.938,310.712,-72.601,-176.722,8.115,148.627
C05006=1169.934,310.960,-72.632,-176.720,8.118,148.627
C05007=1169.930,311.208,-72.663,-176.717,8.121,148.627
C05008=1169.925,311.456,-72.694,-176.715,8.124,148.627
C05009=1169.921,311.704,-72.726,-176.712,8.127,148.627
C05010=1169.917,311.952,-72.757,-176.710,8.130,148.628
C05011=1169.913,312.201,-72.788,-176.707,8.133,148.628
C05012=1169.908,312.448,-72.819,-176.705,8.137,148.628
C05013=1169.904,312.696,-72.850,-176.702,8.140,148.628
C05014=1169.900,312.945,-72.881,-176.699,8.144,148.628
C05015=1169.895,313.192,-72.913,-176.697,8.147,148.628
C05016=1169.891,313.441,-72.944,-176.694,8.150,148.628
C05017=1169.887,313.717,-72.978,-176.692,8.153,148.628
C05018=1169.882,313.994,-73.014,-176.688,8.157,148.628
C05019=1169.877,314.272,-73.048,-176.686,8.160,148.628
C05020=1169.873,314.548,-73.083,-176.683,8.164,148.628
C05021=1169.869,314.796,-73.115,-176.680,8.167,148.629
C05022=1169.864,315.044,-73.146,-176.678,8.170,148.629
C05023=1169.860,315.292,-73.178,-176.675,8.174,148.629
C05024=1169.856,315.540,-73.209,-176.673,8.177,148.629
C05025=1169.852,315.788,-73.241,-176.670,8.180,148.629
C05026=1169.847,316.036,-73.271,-176.668,8.183,148.629
C05027=1169.844,316.284,-73.303,-176.665,8.186,148.629
C05028=1169.839,316.532,-73.335,-176.663,8.189,148.629
C05029=1169.835,316.780,-73.366,-176.660,8.192,148.629
C05030=1169.832,317.029,-73.398,-176.658,8.195,148.629
C05031=1169.827,317.276,-73.428,-176.655,8.199,148.629
C05032=1169.823,317.525,-73.460,-176.652,8.202,148.629
C05033=1169.819,317.772,-73.492,-176.650,8.206,148.630
C05034=1169.815,318.021,-73.523,-176.647,8.209,148.630
C05035=1169.810,318.268,-73.555,-176.645,8.212,148.630
C05036=1169.806,318.516,-73.587,-176.642,8.215,148.630
C05037=1169.802,318.764,-73.618,-176.640,8.218,148.630
C05038=1169.798,319.012,-73.649,-176.637,8.222,148.630
C05039=1169.794,319.260,-73.681,-176.635,8.225,148.630
C05040=1169.790,319.508,-73.713,-176.632,8.228,148.630
C05041=1169.785,319.756,-73.745,-176.630,8.231,148.630
C05042=1169.781,320.004,-73.776,-176.627,8.234,148.631
C05043=1169.777,320.252,-73.808,-176.625,8.237,148.631
C05044=1169.773,320.500,-73.840,-176.622,8.240,148.631
C05045=1169.769,320.747,-73.871,-176.620,8.244,148.631
C05046=1169.765,320.996,-73.904,-176.617,8.248,148.631
C05047=1169.761,321.244,-73.935,-176.614,8.251,148.631
C05048=1169.756,321.492,-73.966,-176.612,8.254,148.631
C05049=1169.753,321.740,-73.998,-176.609,8.257,148.631
C05050=1169.748,321.987,-74.030,-176.607,8.260,148.631
C05051=1169.744,322.235,-74.062,-176.604,8.263,148.632
C05052=1169.740,322.483,-74.094,-176.602,8.267,148.632
C05053=1169.736,322.731,-74.125,-176.599,8.270,148.632
C05054=1169.731,322.979,-74.158,-176.597,8.273,148.632
C05055=1169.728,323.227,-74.189,-176.594,8.276,148.632
C05056=1169.723,323.474,-74.221,-176.592,8.279,148.632
C05057=1169.719,323.723,-74.253,-176.589,8.283,148.632
C05058=1169.715,323.971,-74.285,-176.586,8.286,148.632
C05059=1169.711,324.218,-74.317,-176.584,8.290,148.633
C05060=1169.706,324.467,-74.349,-176.582,8.293,148.633
C05061=1169.703,324.715,-74.381,-176.579,8.296,148.633
C05062=1169.699,324.963,-74.413,-176.577,8.299,148.633
C05063=1169.694,325.210,-74.445,-176.574,8.302,148.633
C05064=1169.690,325.458,-74.477,-176.572,8.306,148.633
C05065=1169.686,325.707,-74.509,-176.570,8.309,148.633
C05066=1169.682,325.954,-74.541,-176.566,8.313,148.633
C05067=1169.678,326.202,-74.573,-176.564,8.316,148.634
C05068=1169.674,326.450,-74.606,-176.562,8.319,148.634
C05069=1169.670,326.698,-74.638,-176.559,8.322,148.634
C05070=1169.665,326.945,-74.670,-176.557,8.326,148.634
C05071=1169.661,327.193,-74.701,-176.554,8.329,148.634
C05072=1169.657,327.442,-74.734,-176.552,8.332,148.634
C05073=1169.653,327.690,-74.766,-176.549,8.335,148.634
C05074=1169.648,327.937,-74.799,-176.547,8.338,148.635
C05075=1169.645,328.185,-74.830,-176.544,8.342,148.635
C05076=1169.640,328.433,-74.863,-176.541,8.345,148.635
C05077=1169.636,328.681,-74.895,-176.539,8.349,148.635
C05078=1169.632,328.929,-74.928,-176.536,8.352,148.635
C05079=1169.628,329.176,-74.959,-176.534,8.355,148.635
C05080=1169.624,329.425,-74.992,-176.532,8.358,148.635
C05081=1169.620,329.672,-75.024,-176.530,8.362,148.636
C05082=1169.616,329.921,-75.057,-176.527,8.365,148.636
C05083=1169.612,330.169,-75.089,-176.524,8.369,148.636
C05084=1169.607,330.416,-75.121,-176.522,8.372,148.636
C05085=1169.604,330.664,-75.153,-176.519,8.375,148.636
C05086=1169.599,330.912,-75.186,-176.517,8.378,148.636
C05087=1169.595,331.160,-75.219,-176.514,8.382,148.637
C05088=1169.591,331.408,-75.251,-176.512,8.385,148.637
C05089=1169.587,331.655,-75.283,-176.509,8.388,148.637
C05090=1169.583,331.903,-75.315,-176.507,8.392,148.637
C05091=1169.578,332.151,-75.348,-176.504,8.395,148.637
C05092=1169.574,332.399,-75.381,-176.502,8.399,148.637
C05093=1169.571,332.647,-75.413,-176.499,8.402,148.637
C05094=1169.566,332.895,-75.446,-176.497,8.405,148.638
C05095=1169.562,333.143,-75.478,-176.495,8.408,148.638
C05096=1169.559,333.390,-75.511,-176.492,8.412,148.638
C05097=1169.554,333.638,-75.543,-176.489,8.415,148.638
C05098=1169.549,333.886,-75.576,-176.487,8.419,148.638
C05099=1169.546,334.134,-75.608,-176.485,8.422,148.638
C05100=1169.542,334.382,-75.641,-176.482,8.425,148.639
C05101=1169.537,334.629,-75.674,-176.480,8.429,148.639
C05102=1169.534,334.877,-75.706,-176.477,8.431,148.639
C05103=1169.530,335.125,-75.739,-176.474,8.436,148.639
C05104=1169.525,335.373,-75.772,-176.472,8.439,148.639
C05105=1169.521,335.621,-75.805,-176.470,8.442,148.640
C05106=1169.518,335.869,-75.837,-176.468,8.446,148.640
C05107=1169.513,336.117,-75.870,-176.465,8.448,148.640
C05108=1169.508,336.364,-75.903,-176.462,8.452,148.640
C05109=1169.504,336.612,-75.936,-176.460,8.456,148.640
C05110=1169.501,336.859,-75.968,-176.457,8.459,148.640
C05111=1169.496,337.107,-76.001,-176.455,8.463,148.641
C05112=1169.492,337.355,-76.034,-176.453,8.466,148.641
C05113=1169.488,337.603,-76.067,-176.450,8.469,148.641
C05114=1169.484,337.851,-76.100,-176.447,8.473,148.641
C05115=1169.480,338.099,-76.132,-176.445,8.476,148.641
C05116=1169.476,338.346,-76.165,-176.443,8.480,148.642
C05117=1169.472,338.594,-76.198,-176.440,8.483,148.642
C05118=1169.468,338.842,-76.232,-176.438,8.486,148.642
C05119=1169.464,339.090,-76.265,-176.436,8.489,148.642
C05120=1169.459,339.338,-76.297,-176.432,8.493,148.642
C05121=1169.455,339.617,-76.334,-176.430,8.497,148.642
C05122=1169.451,339.897,-76.372,-176.427,8.501,148.643
C05123=1169.446,340.176,-76.409,-176.424,8.505,148.643
C05124=1169.441,340.455,-76.446,-176.422,8.509,148.643
C05125=1169.437,340.703,-76.480,-176.419,8.512,148.643
C05126=1169.433,340.951,-76.513,-176.417,8.515,148.644
C05127=1169.429,341.198,-76.546,-176.415,8.519,148.644
C05128=1169.425,341.446,-76.579,-176.412,8.522,148.644
C05129=1169.420,341.694,-76.612,-176.409,8.526,148.644
C05130=1169.416,341.942,-76.645,-176.407,8.529,148.644
C05131=1169.412,342.189,-76.678,-176.405,8.532,148.644
C05132=1169.408,342.437,-76.712,-176.402,8.536,148.645
C05133=1169.404,342.686,-76.745,-176.400,8.539,148.645
C05134=1169.400,342.933,-76.778,-176.397,8.543,148.645
C05135=1169.396,343.181,-76.811,-176.395,8.546,148.645
C05136=1169.392,343.429,-76.845,-176.393,8.550,148.646
C05137=1169.388,343.676,-76.878,-176.390,8.553,148.646
C05138=1169.384,343.924,-76.911,-176.388,8.556,148.646
C05139=1169.380,344.172,-76.944,-176.385,8.561,148.646
C05140=1169.375,344.420,-76.977,-176.383,8.564,148.646
C05141=1169.371,344.667,-77.010,-176.381,8.567,148.647
C05142=1169.367,344.914,-77.044,-176.378,8.570,148.647
C05143=1169.363,345.162,-77.077,-176.375,8.575,148.647
C05144=1169.360,345.411,-77.111,-176.373,8.578,148.647
C05145=1169.356,345.658,-77.144,-176.371,8.581,148.648
C05146=1169.352,345.906,-77.177,-176.369,8.584,148.648
C05147=1169.348,346.153,-77.211,-176.366,8.589,148.648
C05148=1169.343,346.401,-77.245,-176.363,8.592,148.648
C05149=1169.339,346.649,-77.278,-176.361,8.595,148.649
C05150=1169.335,346.897,-77.311,-176.359,8.598,148.649
C05151=1169.331,347.144,-77.345,-176.357,8.602,148.649
C05152=1169.327,347.392,-77.379,-176.354,8.606,148.649
C05153=1169.323,347.640,-77.412,-176.351,8.609,148.649
C05154=1169.319,347.887,-77.446,-176.349,8.612,148.650
C05155=1169.314,348.135,-77.479,-176.347,8.616,148.650
C05156=1169.310,348.383,-77.513,-176.344,8.620,148.650
C05157=1169.307,348.631,-77.547,-176.342,8.623,148.651
C05158=1169.303,348.878,-77.580,-176.340,8.627,148.651
C05159=1169.299,349.126,-77.613,-176.338,8.630,148.651
C05160=1169.294,349.374,-77.648,-176.335,8.634,148.651
C05161=1169.290,349.621,-77.681,-176.332,8.637,148.651
C05162=1169.287,349.869,-77.715,-176.330,8.641,148.652
C05163=1169.283,350.117,-77.748,-176.328,8.644,148.652
C05164=1169.278,350.365,-77.782,-176.325,8.648,148.652
C05165=1169.274,350.612,-77.816,-176.323,8.651,148.652
C05166=1169.270,350.860,-77.849,-176.321,8.655,148.653
C05167=1169.267,351.107,-77.883,-176.318,8.659,148.653
C05168=1169.262,351.356,-77.917,-176.316,8.663,148.653
C05169=1169.258,351.603,-77.951,-176.313,8.666,148.653
C05170=1169.255,351.850,-77.985,-176.311,8.669,148.654
C05171=1169.250,352.098,-78.019,-176.308,8.673,148.654
C05172=1169.246,352.346,-78.053,-176.306,8.677,148.654
C05173=1169.242,352.593,-78.086,-176.304,8.680,148.655
C05174=1169.238,352.841,-78.121,-176.302,8.683,148.655
C05175=1169.234,353.089,-78.154,-176.299,8.688,148.655
C05176=1169.230,353.336,-78.188,-176.297,8.691,148.655
C05177=1169.226,353.584,-78.222,-176.294,8.694,148.655
C05178=1169.222,353.832,-78.256,-176.292,8.699,148.656
C05179=1169.217,354.080,-78.290,-176.290,8.702,148.656
C05180=1169.213,354.327,-78.324,-176.287,8.705,148.656
C05181=1169.210,354.575,-78.357,-176.285,8.708,148.657
C05182=1169.205,354.822,-78.392,-176.283,8.713,148.657
C05183=1169.201,355.070,-78.426,-176.280,8.716,148.657
C05184=1169.197,355.318,-78.461,-176.278,8.720,148.658
C05185=1169.193,355.565,-78.494,-176.275,8.724,148.658
C05186=1169.189,355.813,-78.528,-176.273,8.727,148.658
C05187=1169.185,356.061,-78.562,-176.271,8.731,148.658
C05188=1169.182,356.308,-78.596,-176.268,8.735,148.659
C05189=1169.177,356.557,-78.630,-176.266,8.738,148.659
C05190=1169.174,356.804,-78.664,-176.264,8.742,148.659
C05191=1169.169,357.051,-78.699,-176.261,8.746,148.660
C05192=1169.166,357.299,-78.733,-176.259,8.749,148.660
C05193=1169.161,357.546,-78.767,-176.257,8.753,148.660
C05194=1169.157,357.793,-78.801,-176.255,8.756,148.660
C05195=1169.153,358.042,-78.836,-176.252,8.760,148.661
C05196=1169.149,358.289,-78.869,-176.250,8.764,148.661
C05197=1169.145,358.537,-78.904,-176.248,8.767,148.661
C05198=1169.141,358.784,-78.938,-176.245,8.771,148.662
C05199=1169.137,359.032,-78.973,-176.243,8.775,148.662
C05200=1169.134,359.280,-79.007,-176.241,8.778,148.662
C05201=1169.129,359.527,-79.041,-176.239,8.782,148.663
C05202=1169.125,359.775,-79.076,-176.236,8.786,148.663
C05203=1169.121,360.022,-79.110,-176.234,8.789,148.663
C05204=1169.117,360.270,-79.145,-176.232,8.793,148.664
C05205=1169.113,360.518,-79.179,-176.229,8.797,148.664
C05206=1169.109,360.766,-79.213,-176.227,8.800,148.664
C05207=1169.106,361.013,-79.247,-176.225,8.804,148.665
C05208=1169.102,361.261,-79.282,-176.223,8.808,148.665
C05209=1169.097,361.508,-79.317,-176.220,8.811,148.665
C05210=1169.094,361.755,-79.351,-176.218,8.816,148.666
C05211=1169.090,362.003,-79.386,-176.216,8.819,148.666
C05212=1169.085,362.250,-79.421,-176.214,8.823,148.666
C05213=1169.082,362.498,-79.455,-176.211,8.827,148.667
C05214=1169.077,362.746,-79.489,-176.209,8.830,148.667
C05215=1169.073,362.994,-79.524,-176.207,8.834,148.667
C05216=1169.069,363.241,-79.558,-176.204,8.838,148.668
C05217=1169.066,363.488,-79.593,-176.203,8.842,148.668
C05218=1169.061,363.736,-79.628,-176.200,8.845,148.668
C05219=1169.058,363.984,-79.662,-176.198,8.849,148.669
C05220=1169.054,364.232,-79.697,-176.196,8.853,148.669
C05221=1169.050,364.478,-79.732,-176.194,8.856,148.670
C05222=1169.046,364.727,-79.767,-176.192,8.860,148.670
C05223=1169.042,364.974,-79.801,-176.189,8.864,148.670
C05224=1169.038,365.222,-79.836,-176.188,8.868,148.671
C05225=1169.033,365.503,-79.875,-176.185,8.872,148.671
C05226=1169.029,365.786,-79.915,-176.183,8.877,148.672
C05227=1169.025,366.068,-79.955,-176.180,8.880,148.672
C05228=1169.020,366.350,-79.994,-176.178,8.885,148.673
C05229=1169.016,366.598,-80.029,-176.176,8.888,148.673
C05230=1169.012,366.845,-80.065,-176.174,8.893,148.673
C05231=1169.007,367.093,-80.099,-176.172,8.896,148.674
C05232=1169.005,367.340,-80.134,-176.170,8.900,148.674
C05233=1169.000,367.587,-80.169,-176.168,8.903,148.675
C05234=1168.996,367.836,-80.203,-176.166,8.908,148.675
C05235=1168.992,368.082,-80.239,-176.164,8.911,148.676
C05236=1168.988,368.331,-80.273,-176.162,8.915,148.676
C05237=1168.984,368.578,-80.309,-176.160,8.919,148.676
C05238=1168.980,368.825,-80.343,-176.158,8.922,148.677
C05239=1168.977,369.073,-80.378,-176.157,8.926,148.677
C05240=1168.972,369.320,-80.413,-176.155,8.929,148.678
C05241=1168.968,369.568,-80.448,-176.153,8.934,148.678
C05242=1168.964,369.816,-80.483,-176.151,8.938,148.679
C05243=1168.960,370.062,-80.518,-176.149,8.941,148.679
C05244=1168.956,370.311,-80.553,-176.147,8.945,148.680
C05245=1168.953,370.558,-80.589,-176.146,8.949,148.680
C05246=1168.948,370.806,-80.623,-176.144,8.953,148.681
C05247=1168.944,371.053,-80.659,-176.142,8.956,148.681
C05248=1168.941,371.301,-80.694,-176.140,8.960,148.682
C05249=1168.936,371.548,-80.729,-176.139,8.964,148.682
C05250=1168.932,371.795,-80.764,-176.137,8.967,148.683
C05251=1168.928,372.044,-80.799,-176.135,8.971,148.683
C05252=1168.924,372.290,-80.834,-176.134,8.975,148.684
C05253=1168.920,372.538,-80.870,-176.132,8.979,148.684
C05254=1168.917,372.786,-80.905,-176.130,8.982,148.685
C05255=1168.912,373.033,-80.940,-176.129,8.986,148.685
C05256=1168.909,373.280,-80.975,-176.127,8.990,148.686
C05257=1168.905,373.528,-81.011,-176.126,8.994,148.686
C05258=1168.900,373.775,-81.045,-176.124,8.997,148.687
C05259=1168.897,374.023,-81.081,-176.122,9.001,148.688
C05260=1168.893,374.270,-81.117,-176.121,9.005,148.688
C05261=1168.889,374.518,-81.152,-176.119,9.009,148.689
C05262=1168.885,374.765,-81.187,-176.118,9.013,148.689
C05263=1168.881,375.013,-81.222,-176.117,9.016,148.690
C05264=1168.877,375.260,-81.258,-176.115,9.019,148.690
C05265=1168.873,375.507,-81.293,-176.114,9.023,148.691
C05266=1168.869,375.755,-81.328,-176.112,9.027,148.691
C05267=1168.866,376.003,-81.363,-176.111,9.031,148.692
C05268=1168.862,376.250,-81.399,-176.110,9.034,148.693
C05269=1168.858,376.497,-81.434,-176.108,9.038,148.693
C05270=1168.853,376.745,-81.470,-176.107,9.042,148.694
C05271=1168.850,376.992,-81.506,-176.105,9.046,148.694
C05272=1168.846,377.240,-81.541,-176.104,9.049,148.695
C05273=1168.841,377.487,-81.576,-176.103,9.053,148.696
C05274=1168.838,377.735,-81.611,-176.102,9.056,148.696
C05275=1168.834,377.982,-81.647,-176.101,9.060,148.697
C05276=1168.830,378.230,-81.682,-176.099,9.063,148.697
C05277=1168.826,378.477,-81.718,-176.099,9.067,148.698
C05278=1168.822,378.724,-81.754,-176.097,9.071,148.699
C05279=1168.818,378.972,-81.789,-176.096,9.075,148.699
C05280=1168.814,379.219,-81.825,-176.095,9.078,148.700
C05281=1168.811,379.467,-81.860,-176.094,9.082,148.701
C05282=1168.806,379.713,-81.895,-176.093,9.085,148.701
C05283=1168.802,379.961,-81.932,-176.092,9.089,148.702
C05284=1168.798,380.209,-81.967,-176.091,9.092,148.703
C05285=1168.795,380.456,-82.003,-176.090,9.095,148.703
C05286=1168.791,380.704,-82.038,-176.089,9.099,148.704
C05287=1168.787,380.951,-82.073,-176.088,9.102,148.705
C05288=1168.782,381.198,-82.110,-176.087,9.106,148.705
C05289=1168.779,381.446,-82.145,-176.087,9.110,148.706
C05290=1168.775,381.693,-82.181,-176.086,9.113,148.707
C05291=1168.771,381.941,-82.216,-176.085,9.117,148.707
C05292=1168.767,382.189,-82.252,-176.084,9.120,148.708
C05293=1168.763,382.436,-82.288,-176.083,9.124,148.709
C05294=1168.759,382.683,-82.323,-176.083,9.127,148.709
C05295=1168.755,382.931,-82.359,-176.082,9.131,148.710
C05296=1168.751,383.178,-82.395,-176.081,9.134,148.711
C05297=1168.748,383.425,-82.431,-176.080,9.137,148.711
C05298=1168.744,383.673,-82.467,-176.079,9.140,148.712
C05299=1168.740,383.919,-82.502,-176.079,9.144,148.713
C05300=1168.735,384.167,-82.538,-176.079,9.147,148.714
C05301=1168.732,384.415,-82.573,-176.078,9.150,148.714
C05302=1168.728,384.662,-82.609,-176.077,9.154,148.715
C05303=1168.724,384.910,-82.645,-176.077,9.157,148.716
C05304=1168.720,385.157,-82.681,-176.076,9.160,148.716
C05305=1168.717,385.405,-82.717,-176.076,9.164,148.717
C05306=1168.712,385.652,-82.753,-176.075,9.167,148.718
C05307=1168.708,385.899,-82.788,-176.075,9.170,148.719
C05308=1168.704,386.147,-82.824,-176.074,9.174,148.719
C05309=1168.700,386.394,-82.861,-176.074,9.177,148.720
C05310=1168.697,386.641,-82.896,-176.073,9.180,148.721
C05311=1168.693,386.889,-82.932,-176.073,9.184,148.722
C05312=1168.688,387.137,-82.968,-176.073,9.186,148.722
C05313=1168.685,387.384,-83.003,-176.072,9.190,148.723
C05314=1168.681,387.631,-83.040,-176.072,9.193,148.724
C05315=1168.676,387.878,-83.076,-176.072,9.195,148.724
C05316=1168.673,388.126,-83.111,-176.072,9.199,148.725
C05317=1168.669,388.373,-83.147,-176.071,9.202,148.726
C05318=1168.665,388.620,-83.183,-176.071,9.205,148.727
C05319=1168.661,388.868,-83.219,-176.071,9.208,148.728
C05320=1168.658,389.115,-83.255,-176.071,9.211,148.728
C05321=1168.654,389.362,-83.291,-176.071,9.214,148.729
C05322=1168.650,389.610,-83.327,-176.071,9.217,148.730
C05323=1168.646,389.857,-83.363,-176.070,9.220,148.730
C05324=1168.642,390.105,-83.399,-176.071,9.223,148.731
C05325=1168.638,390.351,-83.435,-176.070,9.226,148.732
C05326=1168.633,390.599,-83.471,-176.070,9.229,148.733
C05327=1168.630,390.847,-83.506,-176.071,9.231,148.733
C05328=1168.626,391.094,-83.543,-176.070,9.235,148.734
C05329=1168.622,391.379,-83.584,-176.071,9.237,148.735
C05330=1168.618,391.664,-83.626,-176.070,9.241,148.736
C05331=1168.613,391.949,-83.667,-176.070,9.245,148.737
C05332=1168.609,392.234,-83.709,-176.070,9.247,148.738
C05333=1168.604,392.482,-83.745,-176.071,9.250,148.738
C05334=1168.601,392.729,-83.781,-176.071,9.253,148.739
C05335=1168.597,392.976,-83.817,-176.071,9.256,148.740
C05336=1168.592,393.223,-83.853,-176.071,9.259,148.741
C05337=1168.589,393.471,-83.888,-176.071,9.261,148.741
C05338=1168.585,393.718,-83.925,-176.071,9.264,148.742
C05339=1168.581,393.965,-83.960,-176.071,9.266,148.743
C05340=1168.577,394.213,-83.997,-176.071,9.269,148.743
C05341=1168.573,394.460,-84.033,-176.072,9.271,148.744
C05342=1168.569,394.708,-84.069,-176.072,9.274,148.745
C05343=1168.565,394.955,-84.105,-176.072,9.277,148.746
C05344=1168.562,395.202,-84.141,-176.072,9.279,148.747
C05345=1168.558,395.450,-84.178,-176.073,9.282,148.747
C05346=1168.554,395.697,-84.213,-176.073,9.285,148.748
C05347=1168.550,395.945,-84.249,-176.073,9.287,148.749
C05348=1168.546,396.192,-84.286,-176.073,9.290,148.749
C05349=1168.542,396.440,-84.322,-176.073,9.292,148.750
C05350=1168.539,396.686,-84.358,-176.073,9.295,148.751
C05351=1168.534,396.934,-84.394,-176.074,9.297,148.751
C05352=1168.530,397.182,-84.430,-176.075,9.299,148.752
C05353=1168.526,397.429,-84.467,-176.075,9.302,148.753
C05354=1168.523,397.676,-84.502,-176.075,9.305,148.754
C05355=1168.518,397.923,-84.539,-176.075,9.307,148.755
C05356=1168.514,398.170,-84.574,-176.076,9.309,148.755
C05357=1168.510,398.418,-84.611,-176.076,9.311,148.756
C05358=1168.507,398.665,-84.647,-176.076,9.314,148.757
C05359=1168.503,398.912,-84.683,-176.076,9.317,148.757
C05360=1168.499,399.160,-84.719,-176.077,9.318,148.758
C05361=1168.495,399.407,-84.755,-176.077,9.321,148.759
C05362=1168.491,399.654,-84.791,-176.077,9.323,148.759
C05363=1168.487,399.902,-84.827,-176.078,9.325,148.760
C05364=1168.483,400.149,-84.864,-176.078,9.328,148.761
C05365=1168.480,400.397,-84.899,-176.078,9.330,148.761
C05366=1168.476,400.644,-84.936,-176.079,9.332,148.762
C05367=1168.472,400.891,-84.972,-176.079,9.335,148.763
C05368=1168.468,401.139,-85.009,-176.080,9.336,148.763
C05369=1168.464,401.386,-85.044,-176.080,9.339,148.764
C05370=1168.460,401.633,-85.081,-176.080,9.342,148.765
C05371=1168.456,401.881,-85.117,-176.081,9.343,148.766
C05372=1168.452,402.128,-85.153,-176.081,9.346,148.766
C05373=1168.449,402.375,-85.189,-176.082,9.348,148.767
C05374=1168.445,402.623,-85.226,-176.082,9.350,148.768
C05375=1168.441,402.870,-85.261,-176.083,9.352,148.768
C05376=1168.437,403.117,-85.298,-176.083,9.354,148.769
C05377=1168.432,403.365,-85.334,-176.083,9.356,148.770
C05378=1168.429,403.612,-85.371,-176.084,9.359,148.770
C05379=1168.425,403.860,-85.407,-176.084,9.360,148.771
C05380=1168.421,404.107,-85.443,-176.084,9.363,148.772
C05381=1168.417,404.355,-85.479,-176.085,9.365,148.772
C05382=1168.414,404.601,-85.515,-176.085,9.367,148.773
C05383=1168.409,404.849,-85.552,-176.086,9.369,148.774
C05384=1168.406,405.096,-85.588,-176.086,9.371,148.774
C05385=1168.401,405.344,-85.624,-176.086,9.373,148.775
C05386=1168.398,405.591,-85.660,-176.087,9.375,148.775
C05387=1168.394,405.838,-85.697,-176.087,9.377,148.776
C05388=1168.390,406.085,-85.733,-176.087,9.379,148.777
C05389=1168.386,406.333,-85.770,-176.088,9.381,148.777
C05390=1168.382,406.580,-85.805,-176.088,9.383,148.778
C05391=1168.378,406.827,-85.842,-176.089,9.385,148.779
C05392=1168.375,407.075,-85.878,-176.089,9.387,148.779
C05393=1168.371,407.322,-85.914,-176.089,9.389,148.780
C05394=1168.367,407.570,-85.950,-176.090,9.391,148.781
C05395=1168.363,407.817,-85.987,-176.090,9.393,148.781
C05396=1168.358,408.065,-86.023,-176.091,9.395,148.782
C05397=1168.355,408.311,-86.059,-176.091,9.396,148.782
C05398=1168.351,408.559,-86.096,-176.091,9.399,148.783
C05399=1168.347,408.806,-86.132,-176.092,9.400,148.784
C05400=1168.343,409.053,-86.168,-176.092,9.402,148.784
C05401=1168.340,409.301,-86.204,-176.093,9.405,148.785
C05402=1168.336,409.548,-86.241,-176.093,9.406,148.785
C05403=1168.332,409.795,-86.276,-176.094,9.408,148.786
C05404=1168.328,410.043,-86.313,-176.093,9.410,148.787
C05405=1168.324,410.290,-86.350,-176.094,9.412,148.787
C05406=1168.320,410.537,-86.386,-176.095,9.414,148.788
C05407=1168.316,410.785,-86.423,-176.095,9.415,148.788
C05408=1168.312,411.032,-86.458,-176.095,9.418,148.789
C05409=1168.308,411.279,-86.495,-176.096,9.419,148.790
C05410=1168.304,411.527,-86.530,-176.096,9.421,148.790
C05411=1168.300,411.774,-86.567,-176.096,9.423,148.791
C05412=1168.297,412.021,-86.604,-176.097,9.425,148.791
C05413=1168.293,412.269,-86.640,-176.097,9.427,148.792
C05414=1168.289,412.516,-86.677,-176.098,9.428,148.792
C05415=1168.285,412.763,-86.712,-176.098,9.431,148.793
C05416=1168.281,413.010,-86.749,-176.098,9.432,148.794
C05417=1168.277,413.257,-86.785,-176.099,9.434,148.794
C05418=1168.273,413.505,-86.821,-176.099,9.435,148.795
C05419=1168.270,413.752,-86.858,-176.099,9.438,148.795
C05420=1168.265,414.000,-86.894,-176.099,9.439,148.796
C05421=1168.261,414.247,-86.931,-176.100,9.441,148.796
C05422=1168.258,414.494,-86.967,-176.100,9.442,148.797
C05423=1168.253,414.742,-87.003,-176.100,9.445,148.798
C05424=1168.250,414.989,-87.039,-176.101,9.446,148.798
C05425=1168.246,415.236,-87.076,-176.101,9.448,148.799
C05426=1168.242,415.483,-87.112,-176.102,9.450,148.799
C05427=1168.240,415.731,-87.148,-176.101,9.452,148.800
C05428=1168.239,415.979,-87.184,-176.102,9.454,148.800
C05429=1168.238,416.279,-87.228,-176.103,9.455,148.801
C05430=1168.239,416.580,-87.272,-176.103,9.458,148.801
C05431=1168.241,416.880,-87.315,-176.103,9.459,148.802
C05432=1168.245,417.181,-87.358,-176.103,9.462,148.803
C05433=1167.823,417.182,-87.404,-176.106,9.473,148.806
C05434=1167.819,416.879,-87.360,-176.106,9.470,148.806
C05435=1167.818,416.574,-87.316,-176.106,9.469,148.805
C05436=1167.817,416.271,-87.273,-176.106,9.466,148.805
C05437=1167.817,415.967,-87.228,-176.105,9.464,148.804
C05438=1167.819,415.719,-87.192,-176.105,9.463,148.803
C05439=1167.821,415.472,-87.156,-176.105,9.461,148.803
C05440=1167.825,415.225,-87.119,-176.104,9.459,148.802
C05441=1167.829,414.978,-87.083,-176.104,9.457,148.802
C05442=1167.833,414.730,-87.047,-176.103,9.456,148.801
C05443=1167.836,414.483,-87.010,-176.104,9.453,148.801
C05444=1167.841,414.236,-86.974,-176.103,9.452,148.800
C05445=1167.845,413.988,-86.937,-176.103,9.450,148.800
C05446=1167.848,413.742,-86.901,-176.102,9.449,148.799
C05447=1167.853,413.494,-86.865,-176.102,9.447,148.798
C05448=1167.856,413.247,-86.829,-176.101,9.445,148.798
C05449=1167.860,413.000,-86.792,-176.101,9.443,148.797
C05450=1167.865,412.752,-86.756,-176.100,9.441,148.797
C05451=1167.867,412.504,-86.719,-176.101,9.439,148.796
C05452=1167.872,412.256,-86.683,-176.100,9.437,148.795
C05453=1167.875,412.010,-86.647,-176.100,9.436,148.795
C05454=1167.879,411.762,-86.610,-176.099,9.434,148.794
C05455=1167.883,411.515,-86.574,-176.099,9.432,148.794
C05456=1167.887,411.268,-86.537,-176.099,9.430,148.793
C05457=1167.891,411.020,-86.501,-176.098,9.428,148.793
C05458=1167.895,410.773,-86.465,-176.098,9.427,148.792
C05459=1167.899,410.526,-86.428,-176.098,9.424,148.791
C05460=1167.902,410.278,-86.393,-176.097,9.423,148.791
C05461=1167.907,410.031,-86.356,-176.097,9.421,148.790
C05462=1167.910,409.784,-86.320,-176.096,9.419,148.790
C05463=1167.914,409.536,-86.283,-176.096,9.417,148.789
C05464=1167.919,409.289,-86.247,-176.095,9.415,148.788
C05465=1167.922,409.042,-86.211,-176.095,9.414,148.788
C05466=1167.926,408.795,-86.174,-176.095,9.411,148.787
C05467=1167.930,408.547,-86.139,-176.094,9.410,148.787
C05468=1167.934,408.300,-86.102,-176.094,9.408,148.786
C05469=1167.938,408.052,-86.066,-176.093,9.405,148.785
C05470=1167.942,407.805,-86.029,-176.093,9.404,148.785
C05471=1167.945,407.558,-85.994,-176.092,9.402,148.784
C05472=1167.949,407.311,-85.957,-176.092,9.400,148.783
C05473=1167.953,407.064,-85.921,-176.092,9.398,148.783
C05474=1167.957,406.816,-85.884,-176.091,9.396,148.782
C05475=1167.961,406.569,-85.848,-176.091,9.394,148.782
C05476=1167.965,406.321,-85.812,-176.090,9.392,148.781
C05477=1167.969,406.074,-85.775,-176.090,9.390,148.780
